   DATA[2383,13] := 817.9794;
   DATA[2383,14] := 1.0;
   DATA[2383,15] := 2.0;
   DATA[2383,16] := 1.0;
   DATA[2383,17] := 1.0;
   DATA[2383,18] := 1.0;
   DATA[2383,19] := 2.0;
   DATA[2383,20] := 148.808;
   DATA[2383,21] := 155.0372;
   DATA[2383,22] := 1.71262;
   DATA[2383,23] := 858.5875;
   DATA[2383,24] := 2.0;
   DATA[2383,25] := 2.0;
   DATA[2383,26] := 7.874135;
   DATA[2383,27] := 144.1938;
   DATA[2383,28] := 261.7278;
   DATA[2383,29] := 12.11228;
   DATA[2383,30] := 1.725711;
   DATA[2383,31] := 1.28705;
   DATA[2383,32] := 0.7353967;
   DATA[2383,33] := 0.3084265;
   DATA[2383,34] := 2.0;
   DATA[2383,35] := 250.0801;
   DATA[2383,36] := 1.681991;
   DATA[2383,37] := 188.7977;
   DATA[2383,38] := 0.000128152;
   DATA[2383,39] := 1.0;
   DATA[2383,40] := 1.0;
   DATA[2384,0] := 2.655414;
   DATA[2384,1] := 865.8766;
   DATA[2384,2] := 2.0;
   DATA[2384,3] := 2.0;
   DATA[2384,4] := 262.3366;
   DATA[2384,5] := 8.395475;
   DATA[2384,6] := 329.7103;
   DATA[2384,7] := 2.455131;
   DATA[2384,8] := 2.0;
   DATA[2384,9] := 2.0;
   DATA[2384,10] := 2.0;
   DATA[2384,11] := 19.66195;
   DATA[2384,12] := 2.208244;
   DATA[2384,13] := 818.0595;
   DATA[2384,14] := 1.0;
   DATA[2384,15] := 2.0;
   DATA[2384,16] := 1.0;
   DATA[2384,17] := 1.0;
   DATA[2384,18] := 1.0;
   DATA[2384,19] := 2.0;
   DATA[2384,20] := 148.808;
   DATA[2384,21] := 155.0372;
   DATA[2384,22] := 1.713901;
   DATA[2384,23] := 858.5491;
   DATA[2384,24] := 2.0;
   DATA[2384,25] := 2.0;
   DATA[2384,26] := 7.874135;
   DATA[2384,27] := 144.1938;
   DATA[2384,28] := 261.7278;
   DATA[2384,29] := 12.11228;
   DATA[2384,30] := 1.725711;
   DATA[2384,31] := 1.277443;
   DATA[2384,32] := 0.7353967;
   DATA[2384,33] := 0.3084265;
   DATA[2384,34] := 2.0;
   DATA[2384,35] := 250.0801;
   DATA[2384,36] := 1.681991;
   DATA[2384,37] := 188.7977;
   DATA[2384,38] := 0.000128152;
   DATA[2384,39] := 1.0;
   DATA[2384,40] := 1.0;
   DATA[2385,0] := 2.653813;
   DATA[2385,1] := 865.9943;
   DATA[2385,2] := 2.0;
   DATA[2385,3] := 2.0;
   DATA[2385,4] := 262.3366;
   DATA[2385,5] := 8.395475;
   DATA[2385,6] := 329.7103;
   DATA[2385,7] := 2.455131;
   DATA[2385,8] := 2.0;
   DATA[2385,9] := 2.0;
   DATA[2385,10] := 2.0;
   DATA[2385,11] := 19.68436;
   DATA[2385,12] := 2.208244;
   DATA[2385,13] := 818.1796;
   DATA[2385,14] := 1.0;
   DATA[2385,15] := 2.0;
   DATA[2385,16] := 1.0;
   DATA[2385,17] := 1.0;
   DATA[2385,18] := 1.0;
   DATA[2385,19] := 2.0;
   DATA[2385,20] := 148.808;
   DATA[2385,21] := 155.0372;
   DATA[2385,22] := 1.713901;
   DATA[2385,23] := 858.7413;
   DATA[2385,24] := 2.0;
   DATA[2385,25] := 2.0;
   DATA[2385,26] := 7.874135;
   DATA[2385,27] := 144.1938;
   DATA[2385,28] := 261.7278;
   DATA[2385,29] := 12.11228;
   DATA[2385,30] := 1.725711;
   DATA[2385,31] := 1.265147;
   DATA[2385,32] := 0.7353967;
   DATA[2385,33] := 0.3084265;
   DATA[2385,34] := 2.0;
   DATA[2385,35] := 249.984;
   DATA[2385,36] := 1.681991;
   DATA[2385,37] := 188.8138;
   DATA[2385,38] := 0.000128152;
   DATA[2385,39] := 1.0;
   DATA[2385,40] := 1.0;
   DATA[2386,0] := 2.625308;
   DATA[2386,1] := 866.5439;
   DATA[2386,2] := 2.0;
   DATA[2386,3] := 2.0;
   DATA[2386,4] := 262.3366;
   DATA[2386,5] := 8.395475;
   DATA[2386,6] := 329.7103;
   DATA[2386,7] := 2.456284;
   DATA[2386,8] := 2.0;
   DATA[2386,9] := 2.0;
   DATA[2386,10] := 2.0;
   DATA[2386,11] := 19.70357;
   DATA[2386,12] := 2.208244;
   DATA[2386,13] := 818.1796;
   DATA[2386,14] := 1.0;
   DATA[2386,15] := 2.0;
   DATA[2386,16] := 1.0;
   DATA[2386,17] := 1.0;
   DATA[2386,18] := 1.0;
   DATA[2386,19] := 2.0;
   DATA[2386,20] := 148.808;
   DATA[2386,21] := 155.0372;
   DATA[2386,22] := 1.713901;
   DATA[2386,23] := 859.0874;
   DATA[2386,24] := 2.0;
   DATA[2386,25] := 2.0;
   DATA[2386,26] := 7.874135;
   DATA[2386,27] := 144.2451;
   DATA[2386,28] := 261.7278;
   DATA[2386,29] := 12.11228;
   DATA[2386,30] := 1.725711;
   DATA[2386,31] := 1.271935;
   DATA[2386,32] := 0.7353967;
   DATA[2386,33] := 0.3084265;
   DATA[2386,34] := 2.0;
   DATA[2386,35] := 249.984;
   DATA[2386,36] := 1.681991;
   DATA[2386,37] := 188.8939;
   DATA[2386,38] := 0.000128152;
   DATA[2386,39] := 1.0;
   DATA[2386,40] := 1.0;
   DATA[2387,0] := 2.612818;
   DATA[2387,1] := 866.7009;
   DATA[2387,2] := 2.0;
   DATA[2387,3] := 2.0;
   DATA[2387,4] := 262.3366;
   DATA[2387,5] := 8.395475;
   DATA[2387,6] := 329.7103;
   DATA[2387,7] := 2.456284;
   DATA[2387,8] := 2.0;
   DATA[2387,9] := 2.0;
   DATA[2387,10] := 2.0;
   DATA[2387,11] := 19.67796;
   DATA[2387,12] := 2.208244;
   DATA[2387,13] := 818.2598;
   DATA[2387,14] := 1.0;
   DATA[2387,15] := 2.0;
   DATA[2387,16] := 1.0;
   DATA[2387,17] := 1.0;
   DATA[2387,18] := 1.0;
   DATA[2387,19] := 2.0;
   DATA[2387,20] := 148.808;
   DATA[2387,21] := 155.0372;
   DATA[2387,22] := 1.714798;
   DATA[2387,23] := 859.2797;
   DATA[2387,24] := 2.0;
   DATA[2387,25] := 2.0;
   DATA[2387,26] := 7.874135;
   DATA[2387,27] := 144.322;
   DATA[2387,28] := 261.7278;
   DATA[2387,29] := 11.95847;
   DATA[2387,30] := 1.725711;
   DATA[2387,31] := 1.279365;
   DATA[2387,32] := 0.7353967;
   DATA[2387,33] := 0.3084265;
   DATA[2387,34] := 2.0;
   DATA[2387,35] := 249.984;
   DATA[2387,36] := 1.681991;
   DATA[2387,37] := 188.8939;
   DATA[2387,38] := 0.000128152;
   DATA[2387,39] := 1.0;
   DATA[2387,40] := 1.0;
   DATA[2388,0] := 2.610575;
   DATA[2388,1] := 867.0542;
   DATA[2388,2] := 2.0;
   DATA[2388,3] := 2.0;
   DATA[2388,4] := 262.3366;
   DATA[2388,5] := 8.395475;
   DATA[2388,6] := 329.7103;
   DATA[2388,7] := 2.456284;
   DATA[2388,8] := 2.0;
   DATA[2388,9] := 2.0;
   DATA[2388,10] := 2.0;
   DATA[2388,11] := 19.62033;
   DATA[2388,12] := 2.206963;
   DATA[2388,13] := 818.1796;
   DATA[2388,14] := 1.0;
   DATA[2388,15] := 2.0;
   DATA[2388,16] := 1.0;
   DATA[2388,17] := 1.0;
   DATA[2388,18] := 1.0;
   DATA[2388,19] := 2.0;
   DATA[2388,20] := 148.808;
   DATA[2388,21] := 155.0372;
   DATA[2388,22] := 1.715952;
   DATA[2388,23] := 859.1643;
   DATA[2388,24] := 2.0;
   DATA[2388,25] := 2.0;
   DATA[2388,26] := 7.874135;
   DATA[2388,27] := 144.4501;
   DATA[2388,28] := 261.7278;
   DATA[2388,29] := 11.95847;
   DATA[2388,30] := 1.725711;
   DATA[2388,31] := 1.282311;
   DATA[2388,32] := 0.7353967;
   DATA[2388,33] := 0.3084265;
   DATA[2388,34] := 2.0;
   DATA[2388,35] := 249.984;
   DATA[2388,36] := 1.681991;
   DATA[2388,37] := 188.8939;
   DATA[2388,38] := 0.000128152;
   DATA[2388,39] := 1.0;
   DATA[2388,40] := 1.0;
   DATA[2389,0] := 2.600967;
   DATA[2389,1] := 867.2504;
   DATA[2389,2] := 2.0;
   DATA[2389,3] := 2.0;
   DATA[2389,4] := 262.3366;
   DATA[2389,5] := 8.395475;
   DATA[2389,6] := 329.7103;
   DATA[2389,7] := 2.455003;
   DATA[2389,8] := 2.0;
   DATA[2389,9] := 2.0;
   DATA[2389,10] := 2.0;
   DATA[2389,11] := 19.62033;
   DATA[2389,12] := 2.206963;
   DATA[2389,13] := 818.2598;
   DATA[2389,14] := 1.0;
   DATA[2389,15] := 2.0;
   DATA[2389,16] := 1.0;
   DATA[2389,17] := 1.0;
   DATA[2389,18] := 1.0;
   DATA[2389,19] := 2.0;
   DATA[2389,20] := 148.808;
   DATA[2389,21] := 155.0372;
   DATA[2389,22] := 1.717105;
   DATA[2389,23] := 859.3566;
   DATA[2389,24] := 2.0;
   DATA[2389,25] := 2.0;
   DATA[2389,26] := 7.874135;
   DATA[2389,27] := 144.4501;
   DATA[2389,28] := 261.5996;
   DATA[2389,29] := 11.95847;
   DATA[2389,30] := 1.725711;
   DATA[2389,31] := 1.288843;
   DATA[2389,32] := 0.7353967;
   DATA[2389,33] := 0.3084265;
   DATA[2389,34] := 2.0;
   DATA[2389,35] := 249.984;
   DATA[2389,36] := 1.681991;
   DATA[2389,37] := 188.8939;
   DATA[2389,38] := 0.000128152;
   DATA[2389,39] := 1.0;
   DATA[2389,40] := 1.0;
   DATA[2390,0] := 2.600967;
   DATA[2390,1] := 867.2504;
   DATA[2390,2] := 2.0;
   DATA[2390,3] := 2.0;
   DATA[2390,4] := 262.3366;
   DATA[2390,5] := 8.395475;
   DATA[2390,6] := 329.7103;
   DATA[2390,7] := 2.455003;
   DATA[2390,8] := 2.0;
   DATA[2390,9] := 2.0;
   DATA[2390,10] := 2.0;
   DATA[2390,11] := 19.62033;
   DATA[2390,12] := 2.206963;
   DATA[2390,13] := 818.2598;
   DATA[2390,14] := 1.0;
   DATA[2390,15] := 2.0;
   DATA[2390,16] := 1.0;
   DATA[2390,17] := 1.0;
   DATA[2390,18] := 1.0;
   DATA[2390,19] := 2.0;
   DATA[2390,20] := 148.808;
   DATA[2390,21] := 155.0372;
   DATA[2390,22] := 1.717105;
   DATA[2390,23] := 859.3566;
   DATA[2390,24] := 2.0;
   DATA[2390,25] := 2.0;
   DATA[2390,26] := 7.874135;
   DATA[2390,27] := 144.4501;
   DATA[2390,28] := 261.5996;
   DATA[2390,29] := 11.95847;
   DATA[2390,30] := 1.725711;
   DATA[2390,31] := 1.288843;
   DATA[2390,32] := 0.7353967;
   DATA[2390,33] := 0.3084265;
   DATA[2390,34] := 2.0;
   DATA[2390,35] := 249.984;
   DATA[2390,36] := 1.681991;
   DATA[2390,37] := 188.8939;
   DATA[2390,38] := 0.000128152;
   DATA[2390,39] := 1.0;
   DATA[2390,40] := 1.0;
   DATA[2391,0] := 2.578548;
   DATA[2391,1] := 867.2504;
   DATA[2391,2] := 2.0;
   DATA[2391,3] := 2.0;
   DATA[2391,4] := 262.3366;
   DATA[2391,5] := 8.395475;
   DATA[2391,6] := 329.7103;
   DATA[2391,7] := 2.454362;
   DATA[2391,8] := 2.0;
   DATA[2391,9] := 2.0;
   DATA[2391,10] := 2.0;
   DATA[2391,11] := 19.62994;
   DATA[2391,12] := 2.206963;
   DATA[2391,13] := 818.3398;
   DATA[2391,14] := 1.0;
   DATA[2391,15] := 2.0;
   DATA[2391,16] := 1.0;
   DATA[2391,17] := 1.0;
   DATA[2391,18] := 1.0;
   DATA[2391,19] := 2.0;
   DATA[2391,20] := 148.808;
   DATA[2391,21] := 155.0372;
   DATA[2391,22] := 1.717361;
   DATA[2391,23] := 859.5873;
   DATA[2391,24] := 2.0;
   DATA[2391,25] := 2.0;
   DATA[2391,26] := 7.874135;
   DATA[2391,27] := 144.4501;
   DATA[2391,28] := 261.5996;
   DATA[2391,29] := 11.95847;
   DATA[2391,30] := 1.725711;
   DATA[2391,31] := 1.291789;
   DATA[2391,32] := 0.7353967;
   DATA[2391,33] := 0.3084265;
   DATA[2391,34] := 2.0;
   DATA[2391,35] := 250.1602;
   DATA[2391,36] := 1.681991;
   DATA[2391,37] := 188.8939;
   DATA[2391,38] := 0.000128152;
   DATA[2391,39] := 1.0;
   DATA[2391,40] := 1.0;
   DATA[2392,0] := 2.564135;
   DATA[2392,1] := 867.3289;
   DATA[2392,2] := 2.0;
   DATA[2392,3] := 2.0;
   DATA[2392,4] := 262.3366;
   DATA[2392,5] := 8.395475;
   DATA[2392,6] := 329.7103;
   DATA[2392,7] := 2.454362;
   DATA[2392,8] := 2.0;
   DATA[2392,9] := 2.0;
   DATA[2392,10] := 2.0;
   DATA[2392,11] := 19.66835;
   DATA[2392,12] := 2.206963;
   DATA[2392,13] := 818.1396;
   DATA[2392,14] := 1.0;
   DATA[2392,15] := 2.0;
   DATA[2392,16] := 1.0;
   DATA[2392,17] := 1.0;
   DATA[2392,18] := 1.0;
   DATA[2392,19] := 2.0;
   DATA[2392,20] := 148.808;
   DATA[2392,21] := 155.191;
   DATA[2392,22] := 1.718643;
   DATA[2392,23] := 859.5873;
   DATA[2392,24] := 2.0;
   DATA[2392,25] := 2.0;
   DATA[2392,26] := 7.874135;
   DATA[2392,27] := 144.4501;
   DATA[2392,28] := 261.5996;
   DATA[2392,29] := 11.95847;
   DATA[2392,30] := 1.725711;
   DATA[2392,31] := 1.291405;
   DATA[2392,32] := 0.7353967;
   DATA[2392,33] := 0.3084265;
   DATA[2392,34] := 2.0;
   DATA[2392,35] := 250.1602;
   DATA[2392,36] := 1.681991;
   DATA[2392,37] := 188.8939;
   DATA[2392,38] := 0.000128152;
   DATA[2392,39] := 1.0;
   DATA[2392,40] := 1.0;
   DATA[2393,0] := 2.54684;
   DATA[2393,1] := 867.3289;
   DATA[2393,2] := 2.0;
   DATA[2393,3] := 2.0;
   DATA[2393,4] := 262.3366;
   DATA[2393,5] := 8.395475;
   DATA[2393,6] := 329.7103;
   DATA[2393,7] := 2.454362;
   DATA[2393,8] := 2.0;
   DATA[2393,9] := 2.0;
   DATA[2393,10] := 2.0;
   DATA[2393,11] := 19.66835;
   DATA[2393,12] := 2.206963;
   DATA[2393,13] := 818.2197;
   DATA[2393,14] := 1.0;
   DATA[2393,15] := 2.0;
   DATA[2393,16] := 1.0;
   DATA[2393,17] := 1.0;
   DATA[2393,18] := 1.0;
   DATA[2393,19] := 2.0;
   DATA[2393,20] := 148.808;
   DATA[2393,21] := 155.191;
   DATA[2393,22] := 1.718643;
   DATA[2393,23] := 859.395;
   DATA[2393,24] := 2.0;
   DATA[2393,25] := 2.0;
   DATA[2393,26] := 7.874135;
   DATA[2393,27] := 144.4501;
   DATA[2393,28] := 261.5996;
   DATA[2393,29] := 11.95847;
   DATA[2393,30] := 1.725711;
   DATA[2393,31] := 1.283592;
   DATA[2393,32] := 0.7353967;
   DATA[2393,33] := 0.3084265;
   DATA[2393,34] := 2.0;
   DATA[2393,35] := 250.1602;
   DATA[2393,36] := 1.681991;
   DATA[2393,37] := 188.8939;
   DATA[2393,38] := 0.000128152;
   DATA[2393,39] := 1.0;
   DATA[2393,40] := 1.0;
   DATA[2394,0] := 2.533068;
   DATA[2394,1] := 867.3289;
   DATA[2394,2] := 2.0;
   DATA[2394,3] := 2.0;
   DATA[2394,4] := 262.3366;
   DATA[2394,5] := 8.395475;
   DATA[2394,6] := 329.7103;
   DATA[2394,7] := 2.45449;
   DATA[2394,8] := 2.0;
   DATA[2394,9] := 2.0;
   DATA[2394,10] := 2.0;
   DATA[2394,11] := 19.66835;
   DATA[2394,12] := 2.208372;
   DATA[2394,13] := 818.3398;
   DATA[2394,14] := 1.0;
   DATA[2394,15] := 2.0;
   DATA[2394,16] := 1.0;
   DATA[2394,17] := 1.0;
   DATA[2394,18] := 1.0;
   DATA[2394,19] := 2.0;
   DATA[2394,20] := 148.808;
   DATA[2394,21] := 155.191;
   DATA[2394,22] := 1.718643;
   DATA[2394,23] := 859.8564;
   DATA[2394,24] := 2.0;
   DATA[2394,25] := 2.0;
   DATA[2394,26] := 7.874135;
   DATA[2394,27] := 144.4501;
   DATA[2394,28] := 261.5996;
   DATA[2394,29] := 11.95847;
   DATA[2394,30] := 1.725711;
   DATA[2394,31] := 1.273601;
   DATA[2394,32] := 0.7353967;
   DATA[2394,33] := 0.3084265;
   DATA[2394,34] := 2.0;
   DATA[2394,35] := 250.1602;
   DATA[2394,36] := 1.617916;
   DATA[2394,37] := 188.8939;
   DATA[2394,38] := 0.000128152;
   DATA[2394,39] := 1.0;
   DATA[2394,40] := 1.0;
   DATA[2395,0] := 2.516414;
   DATA[2395,1] := 867.3289;
   DATA[2395,2] := 2.0;
   DATA[2395,3] := 2.0;
   DATA[2395,4] := 262.3366;
   DATA[2395,5] := 8.395475;
   DATA[2395,6] := 329.7103;
   DATA[2395,7] := 2.45449;
   DATA[2395,8] := 2.0;
   DATA[2395,9] := 2.0;
   DATA[2395,10] := 2.0;
   DATA[2395,11] := 19.67796;
   DATA[2395,12] := 2.209397;
   DATA[2395,13] := 818.8205;
   DATA[2395,14] := 1.0;
   DATA[2395,15] := 2.0;
   DATA[2395,16] := 1.0;
   DATA[2395,17] := 1.0;
   DATA[2395,18] := 1.0;
   DATA[2395,19] := 2.0;
   DATA[2395,20] := 148.808;
   DATA[2395,21] := 155.191;
   DATA[2395,22] := 1.718643;
   DATA[2395,23] := 859.9718;
   DATA[2395,24] := 2.0;
   DATA[2395,25] := 2.0;
   DATA[2395,26] := 7.874135;
   DATA[2395,27] := 144.4501;
   DATA[2395,28] := 261.5996;
   DATA[2395,29] := 11.95847;
   DATA[2395,30] := 1.725711;
   DATA[2395,31] := 1.264378;
   DATA[2395,32] := 0.7353967;
   DATA[2395,33] := 0.3084265;
   DATA[2395,34] := 2.0;
   DATA[2395,35] := 250.1602;
   DATA[2395,36] := 1.617916;
   DATA[2395,37] := 188.8939;
   DATA[2395,38] := 0.000128152;
   DATA[2395,39] := 1.0;
   DATA[2395,40] := 1.0;
   DATA[2396,0] := 2.503283;
   DATA[2396,1] := 867.3682;
   DATA[2396,2] := 2.0;
   DATA[2396,3] := 2.0;
   DATA[2396,4] := 262.3366;
   DATA[2396,5] := 8.395475;
   DATA[2396,6] := 329.7103;
   DATA[2396,7] := 2.45449;
   DATA[2396,8] := 2.0;
   DATA[2396,9] := 2.0;
   DATA[2396,10] := 2.0;
   DATA[2396,11] := 19.70997;
   DATA[2396,12] := 2.209397;
   DATA[2396,13] := 819.1409;
   DATA[2396,14] := 1.0;
   DATA[2396,15] := 2.0;
   DATA[2396,16] := 1.0;
   DATA[2396,17] := 1.0;
   DATA[2396,18] := 1.0;
   DATA[2396,19] := 2.0;
   DATA[2396,20] := 148.808;
   DATA[2396,21] := 155.191;
   DATA[2396,22] := 1.718643;
   DATA[2396,23] := 859.8564;
   DATA[2396,24] := 2.0;
   DATA[2396,25] := 2.0;
   DATA[2396,26] := 7.874135;
   DATA[2396,27] := 144.4501;
   DATA[2396,28] := 261.5996;
   DATA[2396,29] := 11.95847;
   DATA[2396,30] := 1.725711;
   DATA[2396,31] := 1.261688;
   DATA[2396,32] := 0.7353967;
   DATA[2396,33] := 0.3084265;
   DATA[2396,34] := 2.0;
   DATA[2396,35] := 250.1602;
   DATA[2396,36] := 1.617916;
   DATA[2396,37] := 188.8939;
   DATA[2396,38] := 0.000128152;
   DATA[2396,39] := 1.0;
   DATA[2396,40] := 1.0;
   DATA[2397,0] := 2.481504;
   DATA[2397,1] := 867.2897;
   DATA[2397,2] := 2.0;
   DATA[2397,3] := 2.0;
   DATA[2397,4] := 262.3366;
   DATA[2397,5] := 8.395475;
   DATA[2397,6] := 329.7103;
   DATA[2397,7] := 2.45449;
   DATA[2397,8] := 2.0;
   DATA[2397,9] := 2.0;
   DATA[2397,10] := 2.0;
   DATA[2397,11] := 19.70997;
   DATA[2397,12] := 2.210678;
   DATA[2397,13] := 819.0609;
   DATA[2397,14] := 1.0;
   DATA[2397,15] := 2.0;
   DATA[2397,16] := 1.0;
   DATA[2397,17] := 1.0;
   DATA[2397,18] := 1.0;
   DATA[2397,19] := 2.0;
   DATA[2397,20] := 148.808;
   DATA[2397,21] := 155.191;
   DATA[2397,22] := 1.718643;
   DATA[2397,23] := 859.7795;
   DATA[2397,24] := 2.0;
   DATA[2397,25] := 2.0;
   DATA[2397,26] := 7.874135;
   DATA[2397,27] := 144.4501;
   DATA[2397,28] := 261.5996;
   DATA[2397,29] := 11.95847;
   DATA[2397,30] := 1.725711;
   DATA[2397,31] := 1.267709;
   DATA[2397,32] := 0.7353967;
   DATA[2397,33] := 0.3084265;
   DATA[2397,34] := 2.0;
   DATA[2397,35] := 250.1602;
   DATA[2397,36] := 1.617916;
   DATA[2397,37] := 188.8939;
   DATA[2397,38] := 0.000128152;
   DATA[2397,39] := 1.0;
   DATA[2397,40] := 1.0;
   DATA[2398,0] := 2.469013;
   DATA[2398,1] := 867.5645;
   DATA[2398,2] := 2.0;
   DATA[2398,3] := 2.0;
   DATA[2398,4] := 262.3366;
   DATA[2398,5] := 8.395475;
   DATA[2398,6] := 329.7103;
   DATA[2398,7] := 2.45449;
   DATA[2398,8] := 2.0;
   DATA[2398,9] := 2.0;
   DATA[2398,10] := 2.0;
   DATA[2398,11] := 19.70997;
   DATA[2398,12] := 2.210806;
   DATA[2398,13] := 819.181;
   DATA[2398,14] := 1.0;
   DATA[2398,15] := 2.0;
   DATA[2398,16] := 1.0;
   DATA[2398,17] := 1.0;
   DATA[2398,18] := 1.0;
   DATA[2398,19] := 2.0;
   DATA[2398,20] := 148.808;
   DATA[2398,21] := 155.191;
   DATA[2398,22] := 1.718643;
   DATA[2398,23] := 859.1643;
   DATA[2398,24] := 2.0;
   DATA[2398,25] := 2.0;
   DATA[2398,26] := 7.874135;
   DATA[2398,27] := 144.4501;
   DATA[2398,28] := 261.5996;
   DATA[2398,29] := 11.95847;
   DATA[2398,30] := 1.725711;
   DATA[2398,31] := 1.261688;
   DATA[2398,32] := 0.7353967;
   DATA[2398,33] := 0.3084265;
   DATA[2398,34] := 2.0;
   DATA[2398,35] := 250.1602;
   DATA[2398,36] := 1.617916;
   DATA[2398,37] := 188.8939;
   DATA[2398,38] := 0.000128152;
   DATA[2398,39] := 1.0;
   DATA[2398,40] := 1.0;
   DATA[2399,0] := 2.44243;
   DATA[2399,1] := 866.9756;
   DATA[2399,2] := 2.0;
   DATA[2399,3] := 2.0;
   DATA[2399,4] := 262.3366;
   DATA[2399,5] := 8.395475;
   DATA[2399,6] := 329.7103;
   DATA[2399,7] := 2.45449;
   DATA[2399,8] := 2.0;
   DATA[2399,9] := 2.0;
   DATA[2399,10] := 2.0;
   DATA[2399,11] := 19.70997;
   DATA[2399,12] := 2.210806;
   DATA[2399,13] := 819.5415;
   DATA[2399,14] := 1.0;
   DATA[2399,15] := 2.0;
   DATA[2399,16] := 1.0;
   DATA[2399,17] := 1.0;
   DATA[2399,18] := 1.0;
   DATA[2399,19] := 2.0;
   DATA[2399,20] := 148.808;
   DATA[2399,21] := 155.191;
   DATA[2399,22] := 1.718643;
   DATA[2399,23] := 858.8951;
   DATA[2399,24] := 2.0;
   DATA[2399,25] := 2.0;
   DATA[2399,26] := 7.874135;
   DATA[2399,27] := 144.4501;
   DATA[2399,28] := 261.5996;
   DATA[2399,29] := 11.95847;
   DATA[2399,30] := 1.725968;
   DATA[2399,31] := 1.263866;
   DATA[2399,32] := 0.7353967;
   DATA[2399,33] := 0.3084265;
   DATA[2399,34] := 2.0;
   DATA[2399,35] := 250.0;
   DATA[2399,36] := 1.69801;
   DATA[2399,37] := 188.8939;
   DATA[2399,38] := 0.000128152;
   DATA[2399,39] := 1.0;
   DATA[2399,40] := 1.0;
   DATA[2400,0] := 2.431221;
   DATA[2400,1] := 867.0934;
   DATA[2400,2] := 2.0;
   DATA[2400,3] := 2.0;
   DATA[2400,4] := 262.3366;
   DATA[2400,5] := 8.395475;
   DATA[2400,6] := 329.8129;
   DATA[2400,7] := 2.45449;
   DATA[2400,8] := 2.0;
   DATA[2400,9] := 2.0;
   DATA[2400,10] := 2.0;
   DATA[2400,11] := 19.70997;
   DATA[2400,12] := 2.210806;
   DATA[2400,13] := 819.5815;
   DATA[2400,14] := 1.0;
   DATA[2400,15] := 2.0;
   DATA[2400,16] := 1.0;
   DATA[2400,17] := 1.0;
   DATA[2400,18] := 1.0;
   DATA[2400,19] := 2.0;
   DATA[2400,20] := 148.808;
   DATA[2400,21] := 155.191;
   DATA[2400,22] := 1.718643;
   DATA[2400,23] := 858.972;
   DATA[2400,24] := 2.0;
   DATA[2400,25] := 2.0;
   DATA[2400,26] := 7.874135;
   DATA[2400,27] := 144.4501;
   DATA[2400,28] := 261.5996;
   DATA[2400,29] := 11.95847;
   DATA[2400,30] := 1.726352;
   DATA[2400,31] := 1.271295;
   DATA[2400,32] := 0.7353967;
   DATA[2400,33] := 0.3084265;
   DATA[2400,34] := 2.0;
   DATA[2400,35] := 249.9359;
   DATA[2400,36] := 1.69801;
   DATA[2400,37] := 188.8939;
   DATA[2400,38] := 0.000128152;
   DATA[2400,39] := 1.0;
   DATA[2400,40] := 1.0;
   DATA[2401,0] := 2.428018;
   DATA[2401,1] := 866.6616;
   DATA[2401,2] := 2.0;
   DATA[2401,3] := 2.0;
   DATA[2401,4] := 262.3366;
   DATA[2401,5] := 8.395475;
   DATA[2401,6] := 329.8129;
   DATA[2401,7] := 2.45449;
   DATA[2401,8] := 2.0;
   DATA[2401,9] := 2.0;
   DATA[2401,10] := 2.0;
   DATA[2401,11] := 19.70997;
   DATA[2401,12] := 2.210806;
   DATA[2401,13] := 819.3412;
   DATA[2401,14] := 1.0;
   DATA[2401,15] := 2.0;
   DATA[2401,16] := 1.0;
   DATA[2401,17] := 1.0;
   DATA[2401,18] := 1.0;
   DATA[2401,19] := 2.0;
   DATA[2401,20] := 148.808;
   DATA[2401,21] := 155.191;
   DATA[2401,22] := 1.717233;
   DATA[2401,23] := 858.972;
   DATA[2401,24] := 2.0;
   DATA[2401,25] := 2.0;
   DATA[2401,26] := 7.874135;
   DATA[2401,27] := 144.4501;
   DATA[2401,28] := 261.5996;
   DATA[2401,29] := 11.95847;
   DATA[2401,30] := 1.726352;
   DATA[2401,31] := 1.285001;
   DATA[2401,32] := 0.7353967;
   DATA[2401,33] := 0.3084265;
   DATA[2401,34] := 2.0;
   DATA[2401,35] := 249.9359;
   DATA[2401,36] := 1.69801;
   DATA[2401,37] := 188.8939;
   DATA[2401,38] := 0.000128152;
   DATA[2401,39] := 1.0;
   DATA[2401,40] := 1.0;
   DATA[2402,0] := 2.428018;
   DATA[2402,1] := 866.8579;
   DATA[2402,2] := 2.0;
   DATA[2402,3] := 2.0;
   DATA[2402,4] := 262.3366;
   DATA[2402,5] := 8.395475;
   DATA[2402,6] := 329.8129;
   DATA[2402,7] := 2.45449;
   DATA[2402,8] := 2.0;
   DATA[2402,9] := 2.0;
   DATA[2402,10] := 2.0;
   DATA[2402,11] := 19.70997;
   DATA[2402,12] := 2.210806;
   DATA[2402,13] := 819.7818;
   DATA[2402,14] := 1.0;
   DATA[2402,15] := 2.0;
   DATA[2402,16] := 1.0;
   DATA[2402,17] := 1.0;
   DATA[2402,18] := 1.0;
   DATA[2402,19] := 2.0;
   DATA[2402,20] := 148.808;
   DATA[2402,21] := 155.191;
   DATA[2402,22] := 1.714926;
   DATA[2402,23] := 858.8182;
   DATA[2402,24] := 2.0;
   DATA[2402,25] := 2.0;
   DATA[2402,26] := 7.874135;
   DATA[2402,27] := 144.4501;
   DATA[2402,28] := 261.5996;
   DATA[2402,29] := 11.95847;
   DATA[2402,30] := 1.726224;
   DATA[2402,31] := 1.301012;
   DATA[2402,32] := 0.7353967;
   DATA[2402,33] := 0.3084265;
   DATA[2402,34] := 2.0;
   DATA[2402,35] := 249.9359;
   DATA[2402,36] := 1.69801;
   DATA[2402,37] := 188.6375;
   DATA[2402,38] := 0.000128152;
   DATA[2402,39] := 1.0;
   DATA[2402,40] := 1.0;
   DATA[2403,0] := 2.448836;
   DATA[2403,1] := 866.5439;
   DATA[2403,2] := 2.0;
   DATA[2403,3] := 2.0;
   DATA[2403,4] := 262.3366;
   DATA[2403,5] := 8.395475;
   DATA[2403,6] := 329.8129;
   DATA[2403,7] := 2.455515;
   DATA[2403,8] := 2.0;
   DATA[2403,9] := 2.0;
   DATA[2403,10] := 2.0;
   DATA[2403,11] := 19.71957;
   DATA[2403,12] := 2.210806;
   DATA[2403,13] := 819.8218;
   DATA[2403,14] := 1.0;
   DATA[2403,15] := 2.0;
   DATA[2403,16] := 1.0;
   DATA[2403,17] := 1.0;
   DATA[2403,18] := 1.0;
   DATA[2403,19] := 2.0;
   DATA[2403,20] := 148.808;
   DATA[2403,21] := 155.191;
   DATA[2403,22] := 1.713517;
   DATA[2403,23] := 859.0874;
   DATA[2403,24] := 2.0;
   DATA[2403,25] := 2.0;
   DATA[2403,26] := 7.874135;
   DATA[2403,27] := 144.4501;
   DATA[2403,28] := 261.5996;
   DATA[2403,29] := 11.95847;
   DATA[2403,30] := 1.724942;
   DATA[2403,31] := 1.30178;
   DATA[2403,32] := 0.7353967;
   DATA[2403,33] := 0.3084265;
   DATA[2403,34] := 2.0;
   DATA[2403,35] := 249.8718;
   DATA[2403,36] := 1.69801;
   DATA[2403,37] := 188.6375;
   DATA[2403,38] := 0.000128152;
   DATA[2403,39] := 1.0;
   DATA[2403,40] := 1.0;
   DATA[2404,0] := 2.494315;
   DATA[2404,1] := 866.5439;
   DATA[2404,2] := 2.0;
   DATA[2404,3] := 2.0;
   DATA[2404,4] := 262.3366;
   DATA[2404,5] := 8.395475;
   DATA[2404,6] := 329.8129;
   DATA[2404,7] := 2.456284;
   DATA[2404,8] := 2.0;
   DATA[2404,9] := 2.0;
   DATA[2404,10] := 2.0;
   DATA[2404,11] := 19.76439;
   DATA[2404,12] := 2.210037;
   DATA[2404,13] := 820.1824;
   DATA[2404,14] := 1.0;
   DATA[2404,15] := 2.0;
   DATA[2404,16] := 1.0;
   DATA[2404,17] := 1.0;
   DATA[2404,18] := 1.0;
   DATA[2404,19] := 2.0;
   DATA[2404,20] := 148.808;
   DATA[2404,21] := 155.191;
   DATA[2404,22] := 1.713517;
   DATA[2404,23] := 858.7413;
   DATA[2404,24] := 2.0;
   DATA[2404,25] := 2.0;
   DATA[2404,26] := 7.874135;
   DATA[2404,27] := 144.4501;
   DATA[2404,28] := 261.5996;
   DATA[2404,29] := 11.95847;
   DATA[2404,30] := 1.722892;
   DATA[2404,31] := 1.296401;
   DATA[2404,32] := 0.7353967;
   DATA[2404,33] := 0.3084265;
   DATA[2404,34] := 2.0;
   DATA[2404,35] := 249.7116;
   DATA[2404,36] := 1.69801;
   DATA[2404,37] := 188.6375;
   DATA[2404,38] := 0.000128152;
   DATA[2404,39] := 1.0;
   DATA[2404,40] := 1.0;
   DATA[2405,0] := 2.540115;
   DATA[2405,1] := 866.1121;
   DATA[2405,2] := 2.0;
   DATA[2405,3] := 2.0;
   DATA[2405,4] := 262.3366;
   DATA[2405,5] := 8.395475;
   DATA[2405,6] := 329.8129;
   DATA[2405,7] := 2.456284;
   DATA[2405,8] := 2.0;
   DATA[2405,9] := 2.0;
   DATA[2405,10] := 2.0;
   DATA[2405,11] := 19.76439;
   DATA[2405,12] := 2.208756;
   DATA[2405,13] := 820.2224;
   DATA[2405,14] := 1.0;
   DATA[2405,15] := 2.0;
   DATA[2405,16] := 1.0;
   DATA[2405,17] := 1.0;
   DATA[2405,18] := 1.0;
   DATA[2405,19] := 2.0;
   DATA[2405,20] := 148.808;
   DATA[2405,21] := 155.191;
   DATA[2405,22] := 1.713517;
   DATA[2405,23] := 858.7413;
   DATA[2405,24] := 2.0;
   DATA[2405,25] := 2.0;
   DATA[2405,26] := 7.874135;
   DATA[2405,27] := 144.4501;
   DATA[2405,28] := 261.5996;
   DATA[2405,29] := 11.95847;
   DATA[2405,30] := 1.722892;
   DATA[2405,31] := 1.297682;
   DATA[2405,32] := 0.7353967;
   DATA[2405,33] := 0.3084265;
   DATA[2405,34] := 2.0;
   DATA[2405,35] := 249.7116;
   DATA[2405,36] := 1.69801;
   DATA[2405,37] := 188.6375;
   DATA[2405,38] := 0.000128152;
   DATA[2405,39] := 1.0;
   DATA[2405,40] := 1.0;
   DATA[2406,0] := 2.575986;
   DATA[2406,1] := 865.7981;
   DATA[2406,2] := 2.0;
   DATA[2406,3] := 2.0;
   DATA[2406,4] := 262.3366;
   DATA[2406,5] := 8.395475;
   DATA[2406,6] := 329.6591;
   DATA[2406,7] := 2.456284;
   DATA[2406,8] := 2.0;
   DATA[2406,9] := 2.0;
   DATA[2406,10] := 2.0;
   DATA[2406,11] := 19.76439;
   DATA[2406,12] := 2.208628;
   DATA[2406,13] := 820.3826;
   DATA[2406,14] := 1.0;
   DATA[2406,15] := 2.0;
   DATA[2406,16] := 1.0;
   DATA[2406,17] := 1.0;
   DATA[2406,18] := 1.0;
   DATA[2406,19] := 2.0;
   DATA[2406,20] := 148.808;
   DATA[2406,21] := 155.191;
   DATA[2406,22] := 1.712748;
   DATA[2406,23] := 858.7413;
   DATA[2406,24] := 2.0;
   DATA[2406,25] := 2.0;
   DATA[2406,26] := 7.874135;
   DATA[2406,27] := 144.4501;
   DATA[2406,28] := 261.5996;
   DATA[2406,29] := 11.95847;
   DATA[2406,30] := 1.722892;
   DATA[2406,31] := 1.290509;
   DATA[2406,32] := 0.7353967;
   DATA[2406,33] := 0.3084265;
   DATA[2406,34] := 2.0;
   DATA[2406,35] := 249.7116;
   DATA[2406,36] := 1.69801;
   DATA[2406,37] := 188.6375;
   DATA[2406,38] := 0.000128152;
   DATA[2406,39] := 1.0;
   DATA[2406,40] := 1.0;
   DATA[2407,0] := 2.618582;
   DATA[2407,1] := 865.9943;
   DATA[2407,2] := 2.0;
   DATA[2407,3] := 2.0;
   DATA[2407,4] := 262.3366;
   DATA[2407,5] := 8.394514;
   DATA[2407,6] := 329.6591;
   DATA[2407,7] := 2.456284;
   DATA[2407,8] := 2.0;
   DATA[2407,9] := 2.0;
   DATA[2407,10] := 2.0;
   DATA[2407,11] := 19.7996;
   DATA[2407,12] := 2.205041;
   DATA[2407,13] := 820.4627;
   DATA[2407,14] := 1.0;
   DATA[2407,15] := 2.0;
   DATA[2407,16] := 1.0;
   DATA[2407,17] := 1.0;
   DATA[2407,18] := 1.0;
   DATA[2407,19] := 2.0;
   DATA[2407,20] := 148.808;
   DATA[2407,21] := 155.191;
   DATA[2407,22] := 1.712748;
   DATA[2407,23] := 858.5875;
   DATA[2407,24] := 2.0;
   DATA[2407,25] := 2.0;
   DATA[2407,26] := 7.874135;
   DATA[2407,27] := 144.4501;
   DATA[2407,28] := 261.5996;
   DATA[2407,29] := 11.95847;
   DATA[2407,30] := 1.723148;
   DATA[2407,31] := 1.298962;
   DATA[2407,32] := 0.7353967;
   DATA[2407,33] := 0.3084265;
   DATA[2407,34] := 2.0;
   DATA[2407,35] := 249.7116;
   DATA[2407,36] := 1.69801;
   DATA[2407,37] := 188.6375;
   DATA[2407,38] := 0.000128152;
   DATA[2407,39] := 1.0;
   DATA[2407,40] := 1.0;
   DATA[2408,0] := 2.655735;
   DATA[2408,1] := 865.9943;
   DATA[2408,2] := 2.0;
   DATA[2408,3] := 2.0;
   DATA[2408,4] := 262.3366;
   DATA[2408,5] := 8.394514;
   DATA[2408,6] := 329.6591;
   DATA[2408,7] := 2.456284;
   DATA[2408,8] := 2.0;
   DATA[2408,9] := 2.0;
   DATA[2408,10] := 2.0;
   DATA[2408,11] := 19.80601;
   DATA[2408,12] := 2.205041;
   DATA[2408,13] := 820.2625;
   DATA[2408,14] := 1.0;
   DATA[2408,15] := 2.0;
   DATA[2408,16] := 1.0;
   DATA[2408,17] := 1.0;
   DATA[2408,18] := 1.0;
   DATA[2408,19] := 2.0;
   DATA[2408,20] := 148.808;
   DATA[2408,21] := 155.3448;
   DATA[2408,22] := 1.712748;
   DATA[2408,23] := 858.4337;
   DATA[2408,24] := 2.0;
   DATA[2408,25] := 2.0;
   DATA[2408,26] := 7.874135;
   DATA[2408,27] := 144.4501;
   DATA[2408,28] := 261.5996;
   DATA[2408,29] := 11.95847;
   DATA[2408,30] := 1.724301;
   DATA[2408,31] := 1.292686;
   DATA[2408,32] := 0.7353967;
   DATA[2408,33] := 0.3084265;
   DATA[2408,34] := 2.0;
   DATA[2408,35] := 249.8718;
   DATA[2408,36] := 1.69801;
   DATA[2408,37] := 188.6375;
   DATA[2408,38] := 0.000128152;
   DATA[2408,39] := 1.0;
   DATA[2408,40] := 1.0;
   DATA[2409,0] := 2.658937;
   DATA[2409,1] := 866.4654;
   DATA[2409,2] := 2.0;
   DATA[2409,3] := 2.0;
   DATA[2409,4] := 262.3366;
   DATA[2409,5] := 8.394514;
   DATA[2409,6] := 329.6591;
   DATA[2409,7] := 2.456284;
   DATA[2409,8] := 2.0;
   DATA[2409,9] := 2.0;
   DATA[2409,10] := 2.0;
   DATA[2409,11] := 19.80601;
   DATA[2409,12] := 2.205041;
   DATA[2409,13] := 820.0622;
   DATA[2409,14] := 1.0;
   DATA[2409,15] := 2.0;
   DATA[2409,16] := 1.0;
   DATA[2409,17] := 1.0;
   DATA[2409,18] := 1.0;
   DATA[2409,19] := 2.0;
   DATA[2409,20] := 148.808;
   DATA[2409,21] := 155.3448;
   DATA[2409,22] := 1.714798;
   DATA[2409,23] := 858.2415;
   DATA[2409,24] := 2.0;
   DATA[2409,25] := 2.0;
   DATA[2409,26] := 7.874135;
   DATA[2409,27] := 144.4501;
   DATA[2409,28] := 261.5996;
   DATA[2409,29] := 11.95847;
   DATA[2409,30] := 1.724301;
   DATA[2409,31] := 1.282567;
   DATA[2409,32] := 0.7353967;
   DATA[2409,33] := 0.3084265;
   DATA[2409,34] := 2.0;
   DATA[2409,35] := 249.8718;
   DATA[2409,36] := 1.69801;
   DATA[2409,37] := 188.6856;
   DATA[2409,38] := 0.000128152;
   DATA[2409,39] := 1.0;
   DATA[2409,40] := 1.0;
   DATA[2410,0] := 2.646767;
   DATA[2410,1] := 866.5439;
   DATA[2410,2] := 2.0;
   DATA[2410,3] := 2.0;
   DATA[2410,4] := 262.3366;
   DATA[2410,5] := 8.394514;
   DATA[2410,6] := 329.6591;
   DATA[2410,7] := 2.456284;
   DATA[2410,8] := 2.0;
   DATA[2410,9] := 2.0;
   DATA[2410,10] := 2.0;
   DATA[2410,11] := 19.80601;
   DATA[2410,12] := 2.205041;
   DATA[2410,13] := 820.1423;
   DATA[2410,14] := 1.0;
   DATA[2410,15] := 2.0;
   DATA[2410,16] := 1.0;
   DATA[2410,17] := 1.0;
   DATA[2410,18] := 1.0;
   DATA[2410,19] := 2.0;
   DATA[2410,20] := 148.808;
   DATA[2410,21] := 155.3448;
   DATA[2410,22] := 1.715311;
   DATA[2410,23] := 859.1643;
   DATA[2410,24] := 2.0;
   DATA[2410,25] := 2.0;
   DATA[2410,26] := 7.874135;
   DATA[2410,27] := 144.4501;
   DATA[2410,28] := 261.5996;
   DATA[2410,29] := 11.95847;
   DATA[2410,30] := 1.724301;
   DATA[2410,31] := 1.281286;
   DATA[2410,32] := 0.7353967;
   DATA[2410,33] := 0.3084265;
   DATA[2410,34] := 2.0;
   DATA[2410,35] := 249.8718;
   DATA[2410,36] := 1.69801;
   DATA[2410,37] := 188.7657;
   DATA[2410,38] := 0.000128152;
   DATA[2410,39] := 1.0;
   DATA[2410,40] := 1.0;
   DATA[2411,0] := 2.62723;
   DATA[2411,1] := 866.1906;
   DATA[2411,2] := 2.0;
   DATA[2411,3] := 2.0;
   DATA[2411,4] := 262.3366;
   DATA[2411,5] := 8.394514;
   DATA[2411,6] := 329.6591;
   DATA[2411,7] := 2.456284;
   DATA[2411,8] := 2.0;
   DATA[2411,9] := 2.0;
   DATA[2411,10] := 2.0;
   DATA[2411,11] := 19.7804;
   DATA[2411,12] := 2.205554;
   DATA[2411,13] := 820.1423;
   DATA[2411,14] := 1.0;
   DATA[2411,15] := 2.0;
   DATA[2411,16] := 1.0;
   DATA[2411,17] := 1.0;
   DATA[2411,18] := 1.0;
   DATA[2411,19] := 2.0;
   DATA[2411,20] := 148.808;
   DATA[2411,21] := 155.3448;
   DATA[2411,22] := 1.715824;
   DATA[2411,23] := 859.5104;
   DATA[2411,24] := 2.0;
   DATA[2411,25] := 2.0;
   DATA[2411,26] := 7.874135;
   DATA[2411,27] := 144.4501;
   DATA[2411,28] := 261.5996;
   DATA[2411,29] := 11.95847;
   DATA[2411,30] := 1.724301;
   DATA[2411,31] := 1.281286;
   DATA[2411,32] := 0.7353967;
   DATA[2411,33] := 0.3084265;
   DATA[2411,34] := 2.0;
   DATA[2411,35] := 249.8718;
   DATA[2411,36] := 1.69801;
   DATA[2411,37] := 188.9259;
   DATA[2411,38] := 0.000128152;
   DATA[2411,39] := 1.0;
   DATA[2411,40] := 1.0;
   DATA[2412,0] := 2.619543;
   DATA[2412,1] := 866.3476;
   DATA[2412,2] := 2.0;
   DATA[2412,3] := 2.0;
   DATA[2412,4] := 262.3366;
   DATA[2412,5] := 8.394514;
   DATA[2412,6] := 329.6591;
   DATA[2412,7] := 2.456284;
   DATA[2412,8] := 2.0;
   DATA[2412,9] := 2.0;
   DATA[2412,10] := 2.0;
   DATA[2412,11] := 19.76759;
   DATA[2412,12] := 2.207988;
   DATA[2412,13] := 820.3425;
   DATA[2412,14] := 1.0;
   DATA[2412,15] := 2.0;
   DATA[2412,16] := 1.0;
   DATA[2412,17] := 1.0;
   DATA[2412,18] := 1.0;
   DATA[2412,19] := 2.0;
   DATA[2412,20] := 148.808;
   DATA[2412,21] := 155.3448;
   DATA[2412,22] := 1.715824;
   DATA[2412,23] := 859.8564;
   DATA[2412,24] := 2.0;
   DATA[2412,25] := 2.0;
   DATA[2412,26] := 7.874135;
   DATA[2412,27] := 144.4501;
   DATA[2412,28] := 261.5996;
   DATA[2412,29] := 11.95847;
   DATA[2412,30] := 1.724301;
   DATA[2412,31] := 1.291277;
   DATA[2412,32] := 0.7353967;
   DATA[2412,33] := 0.3084265;
   DATA[2412,34] := 2.0;
   DATA[2412,35] := 250.0;
   DATA[2412,36] := 1.69801;
   DATA[2412,37] := 188.9259;
   DATA[2412,38] := 0.000128152;
   DATA[2412,39] := 1.0;
   DATA[2412,40] := 1.0;
   DATA[2413,0] := 2.614099;
   DATA[2413,1] := 865.9943;
   DATA[2413,2] := 2.0;
   DATA[2413,3] := 2.0;
   DATA[2413,4] := 262.3366;
   DATA[2413,5] := 8.394514;
   DATA[2413,6] := 329.6591;
   DATA[2413,7] := 2.454875;
   DATA[2413,8] := 2.0;
   DATA[2413,9] := 2.0;
   DATA[2413,10] := 2.0;
   DATA[2413,11] := 19.76759;
   DATA[2413,12] := 2.208756;
   DATA[2413,13] := 820.4627;
   DATA[2413,14] := 1.0;
   DATA[2413,15] := 2.0;
   DATA[2413,16] := 1.0;
   DATA[2413,17] := 1.0;
   DATA[2413,18] := 1.0;
   DATA[2413,19] := 2.0;
   DATA[2413,20] := 148.808;
   DATA[2413,21] := 155.3448;
   DATA[2413,22] := 1.715824;
   DATA[2413,23] := 860.2794;
   DATA[2413,24] := 2.0;
   DATA[2413,25] := 2.0;
   DATA[2413,26] := 7.874135;
   DATA[2413,27] := 144.4501;
   DATA[2413,28] := 261.5996;
   DATA[2413,29] := 11.95847;
   DATA[2413,30] := 1.724301;
   DATA[2413,31] := 1.302037;
   DATA[2413,32] := 0.7353967;
   DATA[2413,33] := 0.3084265;
   DATA[2413,34] := 2.0;
   DATA[2413,35] := 250.016;
   DATA[2413,36] := 1.69801;
   DATA[2413,37] := 188.9259;
   DATA[2413,38] := 0.000128152;
   DATA[2413,39] := 1.0;
   DATA[2413,40] := 1.0;
   DATA[2414,0] := 2.60481;
   DATA[2414,1] := 865.9158;
   DATA[2414,2] := 2.0;
   DATA[2414,3] := 2.0;
   DATA[2414,4] := 262.3366;
   DATA[2414,5] := 8.396757;
   DATA[2414,6] := 329.7872;
   DATA[2414,7] := 2.454875;
   DATA[2414,8] := 2.0;
   DATA[2414,9] := 2.0;
   DATA[2414,10] := 2.0;
   DATA[2414,11] := 19.76759;
   DATA[2414,12] := 2.208756;
   DATA[2414,13] := 820.0222;
   DATA[2414,14] := 1.0;
   DATA[2414,15] := 2.0;
   DATA[2414,16] := 1.0;
   DATA[2414,17] := 1.0;
   DATA[2414,18] := 1.0;
   DATA[2414,19] := 2.0;
   DATA[2414,20] := 148.808;
   DATA[2414,21] := 155.3448;
   DATA[2414,22] := 1.717233;
   DATA[2414,23] := 860.4717;
   DATA[2414,24] := 2.0;
   DATA[2414,25] := 2.0;
   DATA[2414,26] := 7.874135;
   DATA[2414,27] := 144.4501;
   DATA[2414,28] := 261.5996;
   DATA[2414,29] := 11.95847;
   DATA[2414,30] := 1.724301;
   DATA[2414,31] := 1.302037;
   DATA[2414,32] := 0.7353967;
   DATA[2414,33] := 0.3084265;
   DATA[2414,34] := 2.0;
   DATA[2414,35] := 250.016;
   DATA[2414,36] := 1.69801;
   DATA[2414,37] := 188.8138;
   DATA[2414,38] := 0.000128152;
   DATA[2414,39] := 1.0;
   DATA[2414,40] := 1.0;
   DATA[2415,0] := 2.579509;
   DATA[2415,1] := 866.1514;
   DATA[2415,2] := 2.0;
   DATA[2415,3] := 2.0;
   DATA[2415,4] := 262.3366;
   DATA[2415,5] := 8.396757;
   DATA[2415,6] := 329.7872;
   DATA[2415,7] := 2.455515;
   DATA[2415,8] := 2.0;
   DATA[2415,9] := 2.0;
   DATA[2415,10] := 2.0;
   DATA[2415,11] := 19.79;
   DATA[2415,12] := 2.209653;
   DATA[2415,13] := 820.5829;
   DATA[2415,14] := 1.0;
   DATA[2415,15] := 2.0;
   DATA[2415,16] := 1.0;
   DATA[2415,17] := 1.0;
   DATA[2415,18] := 1.0;
   DATA[2415,19] := 2.0;
   DATA[2415,20] := 148.808;
   DATA[2415,21] := 155.3448;
   DATA[2415,22] := 1.717361;
   DATA[2415,23] := 860.7024;
   DATA[2415,24] := 2.0;
   DATA[2415,25] := 2.0;
   DATA[2415,26] := 7.874135;
   DATA[2415,27] := 144.5014;
   DATA[2415,28] := 261.5996;
   DATA[2415,29] := 11.95847;
   DATA[2415,30] := 1.726737;
   DATA[2415,31] := 1.302037;
   DATA[2415,32] := 0.7353967;
   DATA[2415,33] := 0.3084265;
   DATA[2415,34] := 2.0;
   DATA[2415,35] := 250.016;
   DATA[2415,36] := 1.69801;
   DATA[2415,37] := 188.8138;
   DATA[2415,38] := 0.000128152;
   DATA[2415,39] := 1.0;
   DATA[2415,40] := 1.0;
   DATA[2416,0] := 2.561573;
   DATA[2416,1] := 866.0729;
   DATA[2416,2] := 2.0;
   DATA[2416,3] := 2.0;
   DATA[2416,4] := 262.3366;
   DATA[2416,5] := 8.396757;
   DATA[2416,6] := 329.7872;
   DATA[2416,7] := 2.456156;
   DATA[2416,8] := 2.0;
   DATA[2416,9] := 2.0;
   DATA[2416,10] := 2.0;
   DATA[2416,11] := 19.83162;
   DATA[2416,12] := 2.209653;
   DATA[2416,13] := 820.4227;
   DATA[2416,14] := 1.0;
   DATA[2416,15] := 2.0;
   DATA[2416,16] := 1.0;
   DATA[2416,17] := 1.0;
   DATA[2416,18] := 1.0;
   DATA[2416,19] := 2.0;
   DATA[2416,20] := 148.808;
   DATA[2416,21] := 155.3448;
   DATA[2416,22] := 1.717361;
   DATA[2416,23] := 860.8947;
   DATA[2416,24] := 2.0;
   DATA[2416,25] := 2.0;
   DATA[2416,26] := 7.874135;
   DATA[2416,27] := 144.527;
   DATA[2416,28] := 261.5996;
   DATA[2416,29] := 11.95847;
   DATA[2416,30] := 1.726737;
   DATA[2416,31] := 1.302037;
   DATA[2416,32] := 0.7353967;
   DATA[2416,33] := 0.3084265;
   DATA[2416,34] := 2.0;
   DATA[2416,35] := 250.1762;
   DATA[2416,36] := 1.890238;
   DATA[2416,37] := 188.8138;
   DATA[2416,38] := 0.000128152;
   DATA[2416,39] := 1.0;
   DATA[2416,40] := 1.0;
   DATA[2417,0] := 2.542036;
   DATA[2417,1] := 866.1906;
   DATA[2417,2] := 2.0;
   DATA[2417,3] := 2.0;
   DATA[2417,4] := 262.3366;
   DATA[2417,5] := 8.396757;
   DATA[2417,6] := 329.7872;
   DATA[2417,7] := 2.456156;
   DATA[2417,8] := 2.0;
   DATA[2417,9] := 2.0;
   DATA[2417,10] := 2.0;
   DATA[2417,11] := 19.84762;
   DATA[2417,12] := 2.209653;
   DATA[2417,13] := 820.7431;
   DATA[2417,14] := 1.0;
   DATA[2417,15] := 2.0;
   DATA[2417,16] := 1.0;
   DATA[2417,17] := 1.0;
   DATA[2417,18] := 1.0;
   DATA[2417,19] := 2.0;
   DATA[2417,20] := 148.808;
   DATA[2417,21] := 155.3448;
   DATA[2417,22] := 1.717361;
   DATA[2417,23] := 860.7024;
   DATA[2417,24] := 2.0;
   DATA[2417,25] := 2.0;
   DATA[2417,26] := 7.874135;
   DATA[2417,27] := 144.527;
   DATA[2417,28] := 261.5996;
   DATA[2417,29] := 11.95847;
   DATA[2417,30] := 1.726737;
   DATA[2417,31] := 1.295888;
   DATA[2417,32] := 0.7353967;
   DATA[2417,33] := 0.3084265;
   DATA[2417,34] := 2.0;
   DATA[2417,35] := 250.1762;
   DATA[2417,36] := 1.826162;
   DATA[2417,37] := 188.8618;
   DATA[2417,38] := 0.000128152;
   DATA[2417,39] := 1.0;
   DATA[2417,40] := 1.0;
   DATA[2418,0] := 2.528264;
   DATA[2418,1] := 866.3083;
   DATA[2418,2] := 2.0;
   DATA[2418,3] := 2.0;
   DATA[2418,4] := 262.3366;
   DATA[2418,5] := 8.396757;
   DATA[2418,6] := 329.7872;
   DATA[2418,7] := 2.456156;
   DATA[2418,8] := 2.0;
   DATA[2418,9] := 2.0;
   DATA[2418,10] := 2.0;
   DATA[2418,11] := 19.84762;
   DATA[2418,12] := 2.209653;
   DATA[2418,13] := 820.3826;
   DATA[2418,14] := 1.0;
   DATA[2418,15] := 2.0;
   DATA[2418,16] := 1.0;
   DATA[2418,17] := 1.0;
   DATA[2418,18] := 1.0;
   DATA[2418,19] := 2.0;
   DATA[2418,20] := 148.808;
   DATA[2418,21] := 155.2935;
   DATA[2418,22] := 1.718771;
   DATA[2418,23] := 861.2407;
   DATA[2418,24] := 2.0;
   DATA[2418,25] := 2.0;
   DATA[2418,26] := 7.874135;
   DATA[2418,27] := 144.527;
   DATA[2418,28] := 261.5996;
   DATA[2418,29] := 11.95847;
   DATA[2418,30] := 1.728659;
   DATA[2418,31] := 1.283079;
   DATA[2418,32] := 0.7353967;
   DATA[2418,33] := 0.3084265;
   DATA[2418,34] := 2.0;
   DATA[2418,35] := 250.1762;
   DATA[2418,36] := 1.762086;
   DATA[2418,37] := 189.006;
   DATA[2418,38] := 0.000128152;
   DATA[2418,39] := 1.0;
   DATA[2418,40] := 1.0;
   DATA[2419,0] := 2.504244;
   DATA[2419,1] := 866.5439;
   DATA[2419,2] := 2.0;
   DATA[2419,3] := 2.0;
   DATA[2419,4] := 262.3366;
   DATA[2419,5] := 8.396757;
   DATA[2419,6] := 329.7872;
   DATA[2419,7] := 2.456156;
   DATA[2419,8] := 2.0;
   DATA[2419,9] := 2.0;
   DATA[2419,10] := 2.0;
   DATA[2419,11] := 19.84762;
   DATA[2419,12] := 2.209653;
   DATA[2419,13] := 820.8232;
   DATA[2419,14] := 1.0;
   DATA[2419,15] := 2.0;
   DATA[2419,16] := 1.0;
   DATA[2419,17] := 1.0;
   DATA[2419,18] := 1.0;
   DATA[2419,19] := 2.0;
   DATA[2419,20] := 148.808;
   DATA[2419,21] := 155.2935;
   DATA[2419,22] := 1.719156;
   DATA[2419,23] := 861.7021;
   DATA[2419,24] := 2.0;
   DATA[2419,25] := 2.0;
   DATA[2419,26] := 7.874135;
   DATA[2419,27] := 144.527;
   DATA[2419,28] := 261.5996;
   DATA[2419,29] := 11.95847;
   DATA[2419,30] := 1.728659;
   DATA[2419,31] := 1.282183;
   DATA[2419,32] := 0.7353967;
   DATA[2419,33] := 0.3084265;
   DATA[2419,34] := 2.0;
   DATA[2419,35] := 250.1762;
   DATA[2419,36] := 1.665972;
   DATA[2419,37] := 189.0381;
   DATA[2419,38] := 0.000128152;
   DATA[2419,39] := 1.0;
   DATA[2419,40] := 1.0;
   DATA[2420,0] := 2.489191;
   DATA[2420,1] := 866.4654;
   DATA[2420,2] := 2.0;
   DATA[2420,3] := 2.0;
   DATA[2420,4] := 262.3366;
   DATA[2420,5] := 8.396757;
   DATA[2420,6] := 329.7872;
   DATA[2420,7] := 2.456156;
   DATA[2420,8] := 2.0;
   DATA[2420,9] := 2.0;
   DATA[2420,10] := 2.0;
   DATA[2420,11] := 19.77079;
   DATA[2420,12] := 2.208756;
   DATA[2420,13] := 820.6229;
   DATA[2420,14] := 1.0;
   DATA[2420,15] := 2.0;
   DATA[2420,16] := 1.0;
   DATA[2420,17] := 1.0;
   DATA[2420,18] := 1.0;
   DATA[2420,19] := 2.0;
   DATA[2420,20] := 148.808;
   DATA[2420,21] := 155.2935;
   DATA[2420,22] := 1.719284;
   DATA[2420,23] := 861.6637;
   DATA[2420,24] := 2.0;
   DATA[2420,25] := 2.0;
   DATA[2420,26] := 7.874135;
   DATA[2420,27] := 144.527;
   DATA[2420,28] := 261.5996;
   DATA[2420,29] := 11.95847;
   DATA[2420,30] := 1.728916;
   DATA[2420,31] := 1.272576;
   DATA[2420,32] := 0.7353967;
   DATA[2420,33] := 0.306761;
   DATA[2420,34] := 2.0;
   DATA[2420,35] := 250.2403;
   DATA[2420,36] := 1.665972;
   DATA[2420,37] := 189.1182;
   DATA[2420,38] := 0.000128152;
   DATA[2420,39] := 1.0;
   DATA[2420,40] := 1.0;
   DATA[2421,0] := 2.471255;
   DATA[2421,1] := 866.5831;
   DATA[2421,2] := 2.0;
   DATA[2421,3] := 2.0;
   DATA[2421,4] := 262.3366;
   DATA[2421,5] := 8.395155;
   DATA[2421,6] := 329.7872;
   DATA[2421,7] := 2.456156;
   DATA[2421,8] := 2.0;
   DATA[2421,9] := 2.0;
   DATA[2421,10] := 2.0;
   DATA[2421,11] := 19.72598;
   DATA[2421,12] := 2.208116;
   DATA[2421,13] := 820.9434;
   DATA[2421,14] := 1.0;
   DATA[2421,15] := 2.0;
   DATA[2421,16] := 1.0;
   DATA[2421,17] := 1.0;
   DATA[2421,18] := 1.0;
   DATA[2421,19] := 2.0;
   DATA[2421,20] := 148.808;
   DATA[2421,21] := 155.2935;
   DATA[2421,22] := 1.720693;
   DATA[2421,23] := 862.202;
   DATA[2421,24] := 2.0;
   DATA[2421,25] := 2.0;
   DATA[2421,26] := 7.874135;
   DATA[2421,27] := 144.527;
   DATA[2421,28] := 261.5996;
   DATA[2421,29] := 11.95847;
   DATA[2421,30] := 1.728916;
   DATA[2421,31] := 1.272064;
   DATA[2421,32] := 0.7353967;
   DATA[2421,33] := 0.306761;
   DATA[2421,34] := 2.0;
   DATA[2421,35] := 250.2724;
   DATA[2421,36] := 1.665972;
   DATA[2421,37] := 189.1182;
   DATA[2421,38] := 0.000128152;
   DATA[2421,39] := 1.0;
   DATA[2421,40] := 1.0;
   DATA[2422,0] := 2.456843;
   DATA[2422,1] := 866.5046;
   DATA[2422,2] := 2.0;
   DATA[2422,3] := 2.0;
   DATA[2422,4] := 262.3366;
   DATA[2422,5] := 8.395155;
   DATA[2422,6] := 329.7872;
   DATA[2422,7] := 2.456156;
   DATA[2422,8] := 2.0;
   DATA[2422,9] := 2.0;
   DATA[2422,10] := 2.0;
   DATA[2422,11] := 19.72598;
   DATA[2422,12] := 2.207091;
   DATA[2422,13] := 820.7831;
   DATA[2422,14] := 1.0;
   DATA[2422,15] := 2.0;
   DATA[2422,16] := 1.0;
   DATA[2422,17] := 1.0;
   DATA[2422,18] := 1.0;
   DATA[2422,19] := 2.0;
   DATA[2422,20] := 148.808;
   DATA[2422,21] := 155.2935;
   DATA[2422,22] := 1.722872;
   DATA[2422,23] := 862.6249;
   DATA[2422,24] := 2.0;
   DATA[2422,25] := 2.0;
   DATA[2422,26] := 7.874135;
   DATA[2422,27] := 144.527;
   DATA[2422,28] := 261.5996;
   DATA[2422,29] := 11.95847;
   DATA[2422,30] := 1.728916;
   DATA[2422,31] := 1.288843;
   DATA[2422,32] := 0.7353967;
   DATA[2422,33] := 0.306761;
   DATA[2422,34] := 2.0;
   DATA[2422,35] := 250.2724;
   DATA[2422,36] := 1.665972;
   DATA[2422,37] := 189.1182;
   DATA[2422,38] := 0.000128152;
   DATA[2422,39] := 1.0;
   DATA[2422,40] := 1.0;
   DATA[2423,0] := 2.456843;
   DATA[2423,1] := 866.5046;
   DATA[2423,2] := 2.0;
   DATA[2423,3] := 2.0;
   DATA[2423,4] := 262.3366;
   DATA[2423,5] := 8.395155;
   DATA[2423,6] := 329.7872;
   DATA[2423,7] := 2.456156;
   DATA[2423,8] := 2.0;
   DATA[2423,9] := 2.0;
   DATA[2423,10] := 2.0;
   DATA[2423,11] := 19.72598;
   DATA[2423,12] := 2.207091;
   DATA[2423,13] := 820.7831;
   DATA[2423,14] := 1.0;
   DATA[2423,15] := 2.0;
   DATA[2423,16] := 1.0;
   DATA[2423,17] := 1.0;
   DATA[2423,18] := 1.0;
   DATA[2423,19] := 2.0;
   DATA[2423,20] := 148.808;
   DATA[2423,21] := 155.2935;
   DATA[2423,22] := 1.722872;
   DATA[2423,23] := 862.6249;
   DATA[2423,24] := 2.0;
   DATA[2423,25] := 2.0;
   DATA[2423,26] := 7.874135;
   DATA[2423,27] := 144.527;
   DATA[2423,28] := 261.5996;
   DATA[2423,29] := 11.95847;
   DATA[2423,30] := 1.728916;
   DATA[2423,31] := 1.288843;
   DATA[2423,32] := 0.7353967;
   DATA[2423,33] := 0.306761;
   DATA[2423,34] := 2.0;
   DATA[2423,35] := 250.2724;
   DATA[2423,36] := 1.665972;
   DATA[2423,37] := 189.1182;
   DATA[2423,38] := 0.000128152;
   DATA[2423,39] := 1.0;
   DATA[2423,40] := 1.0;
   DATA[2424,0] := 2.436345;
   DATA[2424,1] := 866.7794;
   DATA[2424,2] := 2.0;
   DATA[2424,3] := 2.0;
   DATA[2424,4] := 262.3366;
   DATA[2424,5] := 8.395155;
   DATA[2424,6] := 329.7872;
   DATA[2424,7] := 2.453849;
   DATA[2424,8] := 2.0;
   DATA[2424,9] := 2.0;
   DATA[2424,10] := 2.0;
   DATA[2424,11] := 19.70357;
   DATA[2424,12] := 2.20581;
   DATA[2424,13] := 821.0235;
   DATA[2424,14] := 1.0;
   DATA[2424,15] := 2.0;
   DATA[2424,16] := 1.0;
   DATA[2424,17] := 1.0;
   DATA[2424,18] := 1.0;
   DATA[2424,19] := 2.0;
   DATA[2424,20] := 148.808;
   DATA[2424,21] := 155.2935;
   DATA[2424,22] := 1.722872;
   DATA[2424,23] := 862.6634;
   DATA[2424,24] := 2.0;
   DATA[2424,25] := 2.0;
   DATA[2424,26] := 7.874135;
   DATA[2424,27] := 144.527;
   DATA[2424,28] := 261.5996;
   DATA[2424,29] := 11.95847;
   DATA[2424,30] := 1.728916;
   DATA[2424,31] := 1.291789;
   DATA[2424,32] := 0.7353967;
   DATA[2424,33] := 0.306761;
   DATA[2424,34] := 2.0;
   DATA[2424,35] := 250.2724;
   DATA[2424,36] := 1.665972;
   DATA[2424,37] := 189.1182;
   DATA[2424,38] := 0.000128152;
   DATA[2424,39] := 1.0;
   DATA[2424,40] := 1.0;
   DATA[2425,0] := 2.424815;
   DATA[2425,1] := 866.7009;
   DATA[2425,2] := 2.0;
   DATA[2425,3] := 2.0;
   DATA[2425,4] := 262.3366;
   DATA[2425,5] := 8.395155;
   DATA[2425,6] := 329.7872;
   DATA[2425,7] := 2.453721;
   DATA[2425,8] := 2.0;
   DATA[2425,9] := 2.0;
   DATA[2425,10] := 2.0;
   DATA[2425,11] := 19.67476;
   DATA[2425,12] := 2.205426;
   DATA[2425,13] := 821.384;
   DATA[2425,14] := 1.0;
   DATA[2425,15] := 2.0;
   DATA[2425,16] := 1.0;
   DATA[2425,17] := 1.0;
   DATA[2425,18] := 1.0;
   DATA[2425,19] := 2.0;
   DATA[2425,20] := 148.808;
   DATA[2425,21] := 155.3448;
   DATA[2425,22] := 1.722872;
   DATA[2425,23] := 863.2402;
   DATA[2425,24] := 2.0;
   DATA[2425,25] := 2.0;
   DATA[2425,26] := 7.874135;
   DATA[2425,27] := 144.527;
   DATA[2425,28] := 261.5996;
   DATA[2425,29] := 11.95847;
   DATA[2425,30] := 1.726609;
   DATA[2425,31] := 1.291277;
   DATA[2425,32] := 0.7353967;
   DATA[2425,33] := 0.306761;
   DATA[2425,34] := 2.0;
   DATA[2425,35] := 250.2724;
   DATA[2425,36] := 1.665972;
   DATA[2425,37] := 189.1182;
   DATA[2425,38] := 0.000128152;
   DATA[2425,39] := 1.0;
   DATA[2425,40] := 1.0;
   DATA[2426,0] := 2.423213;
   DATA[2426,1] := 866.9364;
   DATA[2426,2] := 2.0;
   DATA[2426,3] := 2.0;
   DATA[2426,4] := 262.3366;
   DATA[2426,5] := 8.395155;
   DATA[2426,6] := 329.7872;
   DATA[2426,7] := 2.453721;
   DATA[2426,8] := 2.0;
   DATA[2426,9] := 2.0;
   DATA[2426,10] := 2.0;
   DATA[2426,11] := 19.70037;
   DATA[2426,12] := 2.205426;
   DATA[2426,13] := 821.4641;
   DATA[2426,14] := 1.0;
   DATA[2426,15] := 2.0;
   DATA[2426,16] := 1.0;
   DATA[2426,17] := 1.0;
   DATA[2426,18] := 1.0;
   DATA[2426,19] := 2.0;
   DATA[2426,20] := 148.808;
   DATA[2426,21] := 155.3448;
   DATA[2426,22] := 1.720565;
   DATA[2426,23] := 863.1633;
   DATA[2426,24] := 2.0;
   DATA[2426,25] := 2.0;
   DATA[2426,26] := 7.874135;
   DATA[2426,27] := 144.527;
   DATA[2426,28] := 261.5996;
   DATA[2426,29] := 11.95847;
   DATA[2426,30] := 1.726609;
   DATA[2426,31] := 1.286922;
   DATA[2426,32] := 0.7353967;
   DATA[2426,33] := 0.306761;
   DATA[2426,34] := 2.0;
   DATA[2426,35] := 250.2724;
   DATA[2426,36] := 1.665972;
   DATA[2426,37] := 189.1182;
   DATA[2426,38] := 0.000128152;
   DATA[2426,39] := 1.0;
   DATA[2426,40] := 1.0;
   DATA[2427,0] := 2.425135;
   DATA[2427,1] := 867.0934;
   DATA[2427,2] := 2.0;
   DATA[2427,3] := 2.0;
   DATA[2427,4] := 262.3366;
   DATA[2427,5] := 8.395155;
   DATA[2427,6] := 329.7872;
   DATA[2427,7] := 2.45308;
   DATA[2427,8] := 2.0;
   DATA[2427,9] := 2.0;
   DATA[2427,10] := 2.0;
   DATA[2427,11] := 19.72277;
   DATA[2427,12] := 2.205426;
   DATA[2427,13] := 821.6643;
   DATA[2427,14] := 1.0;
   DATA[2427,15] := 2.0;
   DATA[2427,16] := 1.0;
   DATA[2427,17] := 1.0;
   DATA[2427,18] := 1.0;
   DATA[2427,19] := 2.0;
   DATA[2427,20] := 148.808;
   DATA[2427,21] := 155.3448;
   DATA[2427,22] := 1.720053;
   DATA[2427,23] := 863.3555;
   DATA[2427,24] := 2.0;
   DATA[2427,25] := 2.0;
   DATA[2427,26] := 7.874135;
   DATA[2427,27] := 144.527;
   DATA[2427,28] := 261.5996;
   DATA[2427,29] := 11.95847;
   DATA[2427,30] := 1.726609;
   DATA[2427,31] := 1.287691;
   DATA[2427,32] := 0.7353967;
   DATA[2427,33] := 0.30785;
   DATA[2427,34] := 2.0;
   DATA[2427,35] := 250.2724;
   DATA[2427,36] := 1.762086;
   DATA[2427,37] := 189.1182;
   DATA[2427,38] := 0.000128152;
   DATA[2427,39] := 1.0;
   DATA[2427,40] := 1.0;
   DATA[2428,0] := 2.461647;
   DATA[2428,1] := 867.2897;
   DATA[2428,2] := 2.0;
   DATA[2428,3] := 2.0;
   DATA[2428,4] := 262.3366;
   DATA[2428,5] := 8.395155;
   DATA[2428,6] := 329.7872;
   DATA[2428,7] := 2.451927;
   DATA[2428,8] := 2.0;
   DATA[2428,9] := 2.0;
   DATA[2428,10] := 2.0;
   DATA[2428,11] := 19.72277;
   DATA[2428,12] := 2.205426;
   DATA[2428,13] := 821.8646;
   DATA[2428,14] := 1.0;
   DATA[2428,15] := 2.0;
   DATA[2428,16] := 1.0;
   DATA[2428,17] := 1.0;
   DATA[2428,18] := 1.0;
   DATA[2428,19] := 2.0;
   DATA[2428,20] := 148.808;
   DATA[2428,21] := 155.3448;
   DATA[2428,22] := 1.720053;
   DATA[2428,23] := 863.1633;
   DATA[2428,24] := 2.0;
   DATA[2428,25] := 2.0;
   DATA[2428,26] := 7.874135;
   DATA[2428,27] := 144.527;
   DATA[2428,28] := 261.5996;
   DATA[2428,29] := 11.95847;
   DATA[2428,30] := 1.726609;
   DATA[2428,31] := 1.287691;
   DATA[2428,32] := 0.7353967;
   DATA[2428,33] := 0.30785;
   DATA[2428,34] := 2.0;
   DATA[2428,35] := 250.2724;
   DATA[2428,36] := 1.762086;
   DATA[2428,37] := 189.1182;
   DATA[2428,38] := 0.000128152;
   DATA[2428,39] := 1.0;
   DATA[2428,40] := 1.0;
   DATA[2429,0] := 2.506806;
   DATA[2429,1] := 867.2897;
   DATA[2429,2] := 2.0;
   DATA[2429,3] := 2.0;
   DATA[2429,4] := 262.3366;
   DATA[2429,5] := 8.395155;
   DATA[2429,6] := 329.7872;
   DATA[2429,7] := 2.451671;
   DATA[2429,8] := 2.0;
   DATA[2429,9] := 2.0;
   DATA[2429,10] := 2.0;
   DATA[2429,11] := 19.72277;
   DATA[2429,12] := 2.205426;
   DATA[2429,13] := 821.9447;
   DATA[2429,14] := 1.0;
   DATA[2429,15] := 2.0;
   DATA[2429,16] := 1.0;
   DATA[2429,17] := 1.0;
   DATA[2429,18] := 1.0;
   DATA[2429,19] := 2.0;
   DATA[2429,20] := 148.808;
   DATA[2429,21] := 155.3448;
   DATA[2429,22] := 1.720053;
   DATA[2429,23] := 863.394;
   DATA[2429,24] := 2.0;
   DATA[2429,25] := 2.0;
   DATA[2429,26] := 7.874135;
   DATA[2429,27] := 144.527;
   DATA[2429,28] := 261.5996;
   DATA[2429,29] := 11.95847;
   DATA[2429,30] := 1.726609;
   DATA[2429,31] := 1.302677;
   DATA[2429,32] := 0.7353967;
   DATA[2429,33] := 0.30785;
   DATA[2429,34] := 2.0;
   DATA[2429,35] := 250.2724;
   DATA[2429,36] := 1.762086;
   DATA[2429,37] := 189.1182;
   DATA[2429,38] := 0.000128152;
   DATA[2429,39] := 1.0;
   DATA[2429,40] := 1.0;
   DATA[2430,0] := 2.550043;
   DATA[2430,1] := 867.1719;
   DATA[2430,2] := 2.0;
   DATA[2430,3] := 2.0;
   DATA[2430,4] := 262.3366;
   DATA[2430,5] := 8.395155;
   DATA[2430,6] := 329.7872;
   DATA[2430,7] := 2.450774;
   DATA[2430,8] := 2.0;
   DATA[2430,9] := 2.0;
   DATA[2430,10] := 2.0;
   DATA[2430,11] := 19.72277;
   DATA[2430,12] := 2.205426;
   DATA[2430,13] := 822.1851;
   DATA[2430,14] := 1.0;
   DATA[2430,15] := 2.0;
   DATA[2430,16] := 1.0;
   DATA[2430,17] := 1.0;
   DATA[2430,18] := 1.0;
   DATA[2430,19] := 2.0;
   DATA[2430,20] := 148.808;
   DATA[2430,21] := 155.3448;
   DATA[2430,22] := 1.720053;
   DATA[2430,23] := 863.2402;
   DATA[2430,24] := 2.0;
   DATA[2430,25] := 2.0;
   DATA[2430,26] := 7.874135;
   DATA[2430,27] := 144.527;
   DATA[2430,28] := 261.5996;
   DATA[2430,29] := 11.95847;
   DATA[2430,30] := 1.726609;
   DATA[2430,31] := 1.307288;
   DATA[2430,32] := 0.7353967;
   DATA[2430,33] := 0.30785;
   DATA[2430,34] := 2.0;
   DATA[2430,35] := 250.2724;
   DATA[2430,36] := 1.762086;
   DATA[2430,37] := 189.1182;
   DATA[2430,38] := 0.000128152;
   DATA[2430,39] := 1.0;
   DATA[2430,40] := 1.0;
   DATA[2431,0] := 2.572783;
   DATA[2431,1] := 866.9756;
   DATA[2431,2] := 2.0;
   DATA[2431,3] := 2.0;
   DATA[2431,4] := 262.3366;
   DATA[2431,5] := 8.395155;
   DATA[2431,6] := 329.7872;
   DATA[2431,7] := 2.450389;
   DATA[2431,8] := 2.0;
   DATA[2431,9] := 2.0;
   DATA[2431,10] := 2.0;
   DATA[2431,11] := 19.75799;
   DATA[2431,12] := 2.207347;
   DATA[2431,13] := 822.3453;
   DATA[2431,14] := 1.0;
   DATA[2431,15] := 2.0;
   DATA[2431,16] := 1.0;
   DATA[2431,17] := 1.0;
   DATA[2431,18] := 1.0;
   DATA[2431,19] := 2.0;
   DATA[2431,20] := 148.808;
   DATA[2431,21] := 155.3448;
   DATA[2431,22] := 1.720053;
   DATA[2431,23] := 863.2402;
   DATA[2431,24] := 2.0;
   DATA[2431,25] := 2.0;
   DATA[2431,26] := 7.874135;
   DATA[2431,27] := 144.527;
   DATA[2431,28] := 261.5996;
   DATA[2431,29] := 11.95847;
   DATA[2431,30] := 1.726609;
   DATA[2431,31] := 1.307288;
   DATA[2431,32] := 0.7353967;
   DATA[2431,33] := 0.3072094;
   DATA[2431,34] := 2.0;
   DATA[2431,35] := 250.2724;
   DATA[2431,36] := 1.762086;
   DATA[2431,37] := 189.1182;
   DATA[2431,38] := 0.000128152;
   DATA[2431,39] := 1.0;
   DATA[2431,40] := 1.0;
   DATA[2432,0] := 2.625308;
   DATA[2432,1] := 867.0542;
   DATA[2432,2] := 2.0;
   DATA[2432,3] := 2.0;
   DATA[2432,4] := 262.3366;
   DATA[2432,5] := 8.395155;
   DATA[2432,6] := 329.7872;
   DATA[2432,7] := 2.451286;
   DATA[2432,8] := 2.0;
   DATA[2432,9] := 2.0;
   DATA[2432,10] := 2.0;
   DATA[2432,11] := 19.77399;
   DATA[2432,12] := 2.208756;
   DATA[2432,13] := 822.2651;
   DATA[2432,14] := 1.0;
   DATA[2432,15] := 2.0;
   DATA[2432,16] := 1.0;
   DATA[2432,17] := 1.0;
   DATA[2432,18] := 1.0;
   DATA[2432,19] := 2.0;
   DATA[2432,20] := 148.808;
   DATA[2432,21] := 155.3448;
   DATA[2432,22] := 1.717233;
   DATA[2432,23] := 863.394;
   DATA[2432,24] := 2.0;
   DATA[2432,25] := 2.0;
   DATA[2432,26] := 7.874135;
   DATA[2432,27] := 144.4501;
   DATA[2432,28] := 261.5996;
   DATA[2432,29] := 11.95847;
   DATA[2432,30] := 1.726609;
   DATA[2432,31] := 1.308057;
   DATA[2432,32] := 0.7353967;
   DATA[2432,33] := 0.3063127;
   DATA[2432,34] := 2.0;
   DATA[2432,35] := 250.2724;
   DATA[2432,36] := 1.665972;
   DATA[2432,37] := 189.1182;
   DATA[2432,38] := 0.000128152;
   DATA[2432,39] := 1.0;
   DATA[2432,40] := 1.0;
   DATA[2433,0] := 2.641322;
   DATA[2433,1] := 867.1327;
   DATA[2433,2] := 2.0;
   DATA[2433,3] := 2.0;
   DATA[2433,4] := 262.3366;
   DATA[2433,5] := 8.395155;
   DATA[2433,6] := 329.7872;
   DATA[2433,7] := 2.451927;
   DATA[2433,8] := 2.0;
   DATA[2433,9] := 2.0;
   DATA[2433,10] := 2.0;
   DATA[2433,11] := 19.77399;
   DATA[2433,12] := 2.208756;
   DATA[2433,13] := 822.2651;
   DATA[2433,14] := 1.0;
   DATA[2433,15] := 2.0;
   DATA[2433,16] := 1.0;
   DATA[2433,17] := 1.0;
   DATA[2433,18] := 1.0;
   DATA[2433,19] := 2.0;
   DATA[2433,20] := 148.808;
   DATA[2433,21] := 155.3448;
   DATA[2433,22] := 1.717233;
   DATA[2433,23] := 863.394;
   DATA[2433,24] := 2.0;
   DATA[2433,25] := 2.0;
   DATA[2433,26] := 7.874135;
   DATA[2433,27] := 144.3732;
   DATA[2433,28] := 261.5996;
   DATA[2433,29] := 11.95847;
   DATA[2433,30] := 1.726609;
   DATA[2433,31] := 1.294351;
   DATA[2433,32] := 0.7353967;
   DATA[2433,33] := 0.3063127;
   DATA[2433,34] := 2.0;
   DATA[2433,35] := 250.3365;
   DATA[2433,36] := 1.665972;
   DATA[2433,37] := 189.1182;
   DATA[2433,38] := 0.000128152;
   DATA[2433,39] := 1.0;
   DATA[2433,40] := 1.0;
   DATA[2434,0] := 2.657016;
   DATA[2434,1] := 867.3682;
   DATA[2434,2] := 2.0;
   DATA[2434,3] := 2.0;
   DATA[2434,4] := 262.3366;
   DATA[2434,5] := 8.395155;
   DATA[2434,6] := 329.7872;
   DATA[2434,7] := 2.451927;
   DATA[2434,8] := 2.0;
   DATA[2434,9] := 2.0;
   DATA[2434,10] := 2.0;
   DATA[2434,11] := 19.68436;
   DATA[2434,12] := 2.208756;
   DATA[2434,13] := 822.4654;
   DATA[2434,14] := 1.0;
   DATA[2434,15] := 2.0;
   DATA[2434,16] := 1.0;
   DATA[2434,17] := 1.0;
   DATA[2434,18] := 1.0;
   DATA[2434,19] := 2.0;
   DATA[2434,20] := 148.808;
   DATA[2434,21] := 155.3448;
   DATA[2434,22] := 1.717233;
   DATA[2434,23] := 863.1633;
   DATA[2434,24] := 2.0;
   DATA[2434,25] := 2.0;
   DATA[2434,26] := 7.874135;
   DATA[2434,27] := 144.3732;
   DATA[2434,28] := 261.5996;
   DATA[2434,29] := 11.95847;
   DATA[2434,30] := 1.726609;
   DATA[2434,31] := 1.292046;
   DATA[2434,32] := 0.7353967;
   DATA[2434,33] := 0.3063127;
   DATA[2434,34] := 2.0;
   DATA[2434,35] := 250.3365;
   DATA[2434,36] := 1.665972;
   DATA[2434,37] := 189.1182;
   DATA[2434,38] := 0.000128152;
   DATA[2434,39] := 1.0;
   DATA[2434,40] := 1.0;
   DATA[2435,0] := 2.657016;
   DATA[2435,1] := 867.5645;
   DATA[2435,2] := 2.0;
   DATA[2435,3] := 2.0;
   DATA[2435,4] := 262.3366;
   DATA[2435,5] := 8.395155;
   DATA[2435,6] := 329.7872;
   DATA[2435,7] := 2.451927;
   DATA[2435,8] := 2.0;
   DATA[2435,9] := 2.0;
   DATA[2435,10] := 2.0;
   DATA[2435,11] := 19.68436;
   DATA[2435,12] := 2.208756;
   DATA[2435,13] := 822.6256;
   DATA[2435,14] := 1.0;
   DATA[2435,15] := 2.0;
   DATA[2435,16] := 1.0;
   DATA[2435,17] := 1.0;
   DATA[2435,18] := 1.0;
   DATA[2435,19] := 2.0;
   DATA[2435,20] := 148.808;
   DATA[2435,21] := 155.3448;
   DATA[2435,22] := 1.715567;
   DATA[2435,23] := 863.2402;
   DATA[2435,24] := 2.0;
   DATA[2435,25] := 2.0;
   DATA[2435,26] := 7.874135;
   DATA[2435,27] := 144.3732;
   DATA[2435,28] := 261.5996;
   DATA[2435,29] := 11.95847;
   DATA[2435,30] := 1.726609;
   DATA[2435,31] := 1.283079;
   DATA[2435,32] := 0.7353967;
   DATA[2435,33] := 0.3074656;
   DATA[2435,34] := 2.0;
   DATA[2435,35] := 250.3365;
   DATA[2435,36] := 1.665972;
   DATA[2435,37] := 189.1182;
   DATA[2435,38] := 0.000128152;
   DATA[2435,39] := 1.0;
   DATA[2435,40] := 1.0;
   DATA[2436,0] := 2.631393;
   DATA[2436,1] := 867.0934;
   DATA[2436,2] := 2.0;
   DATA[2436,3] := 2.0;
   DATA[2436,4] := 262.3366;
   DATA[2436,5] := 8.395155;
   DATA[2436,6] := 329.7872;
   DATA[2436,7] := 2.451927;
   DATA[2436,8] := 2.0;
   DATA[2436,9] := 2.0;
   DATA[2436,10] := 2.0;
   DATA[2436,11] := 19.75799;
   DATA[2436,12] := 2.208756;
   DATA[2436,13] := 822.5455;
   DATA[2436,14] := 1.0;
   DATA[2436,15] := 2.0;
   DATA[2436,16] := 1.0;
   DATA[2436,17] := 1.0;
   DATA[2436,18] := 1.0;
   DATA[2436,19] := 2.0;
   DATA[2436,20] := 148.808;
   DATA[2436,21] := 155.3448;
   DATA[2436,22] := 1.715567;
   DATA[2436,23] := 862.7403;
   DATA[2436,24] := 2.0;
   DATA[2436,25] := 2.0;
   DATA[2436,26] := 7.874135;
   DATA[2436,27] := 144.3732;
   DATA[2436,28] := 261.5996;
   DATA[2436,29] := 11.95847;
   DATA[2436,30] := 1.726609;
   DATA[2436,31] := 1.281542;
   DATA[2436,32] := 0.7353967;
   DATA[2436,33] := 0.3075297;
   DATA[2436,34] := 2.0;
   DATA[2436,35] := 250.016;
   DATA[2436,36] := 1.746067;
   DATA[2436,37] := 188.8939;
   DATA[2436,38] := 0.000128152;
   DATA[2436,39] := 1.0;
   DATA[2436,40] := 1.0;
   DATA[2437,0] := 2.623387;
   DATA[2437,1] := 867.486;
   DATA[2437,2] := 2.0;
   DATA[2437,3] := 2.0;
   DATA[2437,4] := 262.3366;
   DATA[2437,5] := 8.395155;
   DATA[2437,6] := 329.7872;
   DATA[2437,7] := 2.453337;
   DATA[2437,8] := 2.0;
   DATA[2437,9] := 2.0;
   DATA[2437,10] := 2.0;
   DATA[2437,11] := 19.7836;
   DATA[2437,12] := 2.207603;
   DATA[2437,13] := 822.7458;
   DATA[2437,14] := 1.0;
   DATA[2437,15] := 2.0;
   DATA[2437,16] := 1.0;
   DATA[2437,17] := 1.0;
   DATA[2437,18] := 1.0;
   DATA[2437,19] := 2.0;
   DATA[2437,20] := 148.808;
   DATA[2437,21] := 155.3448;
   DATA[2437,22] := 1.715567;
   DATA[2437,23] := 862.8172;
   DATA[2437,24] := 2.0;
   DATA[2437,25] := 2.0;
   DATA[2437,26] := 7.874135;
   DATA[2437,27] := 144.3732;
   DATA[2437,28] := 261.5996;
   DATA[2437,29] := 11.95847;
   DATA[2437,30] := 1.726609;
   DATA[2437,31] := 1.282951;
   DATA[2437,32] := 0.7353967;
   DATA[2437,33] := 0.30785;
   DATA[2437,34] := 2.0;
   DATA[2437,35] := 250.016;
   DATA[2437,36] := 1.746067;
   DATA[2437,37] := 188.8939;
   DATA[2437,38] := 0.000128152;
   DATA[2437,39] := 1.0;
   DATA[2437,40] := 1.0;
   DATA[2438,0] := 2.617942;
   DATA[2438,1] := 867.486;
   DATA[2438,2] := 2.0;
   DATA[2438,3] := 2.0;
   DATA[2438,4] := 262.3366;
   DATA[2438,5] := 8.395155;
   DATA[2438,6] := 329.7872;
   DATA[2438,7] := 2.453337;
   DATA[2438,8] := 2.0;
   DATA[2438,9] := 2.0;
   DATA[2438,10] := 2.0;
   DATA[2438,11] := 19.7836;
   DATA[2438,12] := 2.206322;
   DATA[2438,13] := 822.6657;
   DATA[2438,14] := 1.0;
   DATA[2438,15] := 2.0;
   DATA[2438,16] := 1.0;
   DATA[2438,17] := 1.0;
   DATA[2438,18] := 1.0;
   DATA[2438,19] := 2.0;
   DATA[2438,20] := 148.808;
   DATA[2438,21] := 155.3448;
   DATA[2438,22] := 1.713645;
   DATA[2438,23] := 862.5865;
   DATA[2438,24] := 2.0;
   DATA[2438,25] := 2.0;
   DATA[2438,26] := 7.874135;
   DATA[2438,27] := 144.3732;
   DATA[2438,28] := 261.5996;
   DATA[2438,29] := 11.95847;
   DATA[2438,30] := 1.726609;
   DATA[2438,31] := 1.285129;
   DATA[2438,32] := 0.7353967;
   DATA[2438,33] := 0.3081062;
   DATA[2438,34] := 2.0;
   DATA[2438,35] := 250.016;
   DATA[2438,36] := 1.746067;
   DATA[2438,37] := 188.8939;
   DATA[2438,38] := 0.000128152;
   DATA[2438,39] := 1.0;
   DATA[2438,40] := 1.0;
   DATA[2439,0] := 2.605131;
   DATA[2439,1] := 867.2897;
   DATA[2439,2] := 2.0;
   DATA[2439,3] := 2.0;
   DATA[2439,4] := 262.3366;
   DATA[2439,5] := 8.395155;
   DATA[2439,6] := 329.7872;
   DATA[2439,7] := 2.453337;
   DATA[2439,8] := 2.0;
   DATA[2439,9] := 2.0;
   DATA[2439,10] := 2.0;
   DATA[2439,11] := 19.69396;
   DATA[2439,12] := 2.206322;
   DATA[2439,13] := 822.2651;
   DATA[2439,14] := 1.0;
   DATA[2439,15] := 2.0;
   DATA[2439,16] := 1.0;
   DATA[2439,17] := 1.0;
   DATA[2439,18] := 1.0;
   DATA[2439,19] := 2.0;
   DATA[2439,20] := 148.808;
   DATA[2439,21] := 155.3448;
   DATA[2439,22] := 1.713389;
   DATA[2439,23] := 862.2789;
   DATA[2439,24] := 2.0;
   DATA[2439,25] := 2.0;
   DATA[2439,26] := 7.874135;
   DATA[2439,27] := 144.3732;
   DATA[2439,28] := 261.5996;
   DATA[2439,29] := 11.95847;
   DATA[2439,30] := 1.726609;
   DATA[2439,31] := 1.288075;
   DATA[2439,32] := 0.7353967;
   DATA[2439,33] := 0.3081062;
   DATA[2439,34] := 2.0;
   DATA[2439,35] := 250.016;
   DATA[2439,36] := 1.585878;
   DATA[2439,37] := 188.8939;
   DATA[2439,38] := 0.000128152;
   DATA[2439,39] := 1.0;
   DATA[2439,40] := 1.0;
   DATA[2440,0] := 2.584313;
   DATA[2440,1] := 867.1327;
   DATA[2440,2] := 2.0;
   DATA[2440,3] := 2.0;
   DATA[2440,4] := 262.3366;
   DATA[2440,5] := 8.395155;
   DATA[2440,6] := 329.7103;
   DATA[2440,7] := 2.453337;
   DATA[2440,8] := 2.0;
   DATA[2440,9] := 2.0;
   DATA[2440,10] := 2.0;
   DATA[2440,11] := 19.69396;
   DATA[2440,12] := 2.206322;
   DATA[2440,13] := 822.4254;
   DATA[2440,14] := 1.0;
   DATA[2440,15] := 2.0;
   DATA[2440,16] := 1.0;
   DATA[2440,17] := 1.0;
   DATA[2440,18] := 1.0;
   DATA[2440,19] := 2.0;
   DATA[2440,20] := 148.808;
   DATA[2440,21] := 155.3448;
   DATA[2440,22] := 1.712748;
   DATA[2440,23] := 862.202;
   DATA[2440,24] := 2.0;
   DATA[2440,25] := 2.0;
   DATA[2440,26] := 7.874135;
   DATA[2440,27] := 144.3732;
   DATA[2440,28] := 261.5996;
   DATA[2440,29] := 11.95847;
   DATA[2440,30] := 1.726609;
   DATA[2440,31] := 1.284873;
   DATA[2440,32] := 0.7353967;
   DATA[2440,33] := 0.309003;
   DATA[2440,34] := 2.0;
   DATA[2440,35] := 250.016;
   DATA[2440,36] := 1.585878;
   DATA[2440,37] := 188.8138;
   DATA[2440,38] := 0.000128152;
   DATA[2440,39] := 1.0;
   DATA[2440,40] := 1.0;
   DATA[2441,0] := 2.555488;
   DATA[2441,1] := 867.1719;
   DATA[2441,2] := 2.0;
   DATA[2441,3] := 2.0;
   DATA[2441,4] := 262.3366;
   DATA[2441,5] := 8.395155;
   DATA[2441,6] := 329.6334;
   DATA[2441,7] := 2.453337;
   DATA[2441,8] := 2.0;
   DATA[2441,9] := 2.0;
   DATA[2441,10] := 2.0;
   DATA[2441,11] := 19.69396;
   DATA[2441,12] := 2.206322;
   DATA[2441,13] := 822.1851;
   DATA[2441,14] := 1.0;
   DATA[2441,15] := 2.0;
   DATA[2441,16] := 1.0;
   DATA[2441,17] := 1.0;
   DATA[2441,18] := 1.0;
   DATA[2441,19] := 2.0;
   DATA[2441,20] := 148.808;
   DATA[2441,21] := 155.3448;
   DATA[2441,22] := 1.715952;
   DATA[2441,23] := 861.6252;
   DATA[2441,24] := 2.0;
   DATA[2441,25] := 2.0;
   DATA[2441,26] := 7.874135;
   DATA[2441,27] := 144.3732;
   DATA[2441,28] := 261.5996;
   DATA[2441,29] := 11.95847;
   DATA[2441,30] := 1.726609;
   DATA[2441,31] := 1.282183;
   DATA[2441,32] := 0.7353967;
   DATA[2441,33] := 0.309003;
   DATA[2441,34] := 2.0;
   DATA[2441,35] := 250.016;
   DATA[2441,36] := 1.585878;
   DATA[2441,37] := 188.8138;
   DATA[2441,38] := 0.000128152;
   DATA[2441,39] := 1.0;
   DATA[2441,40] := 1.0;
   DATA[2442,0] := 2.538513;
   DATA[2442,1] := 866.7794;
   DATA[2442,2] := 2.0;
   DATA[2442,3] := 2.0;
   DATA[2442,4] := 262.3366;
   DATA[2442,5] := 8.395155;
   DATA[2442,6] := 329.6334;
   DATA[2442,7] := 2.453337;
   DATA[2442,8] := 2.0;
   DATA[2442,9] := 2.0;
   DATA[2442,10] := 2.0;
   DATA[2442,11] := 19.69396;
   DATA[2442,12] := 2.206322;
   DATA[2442,13] := 822.2651;
   DATA[2442,14] := 1.0;
   DATA[2442,15] := 2.0;
   DATA[2442,16] := 1.0;
   DATA[2442,17] := 1.0;
   DATA[2442,18] := 1.0;
   DATA[2442,19] := 2.0;
   DATA[2442,20] := 148.808;
   DATA[2442,21] := 155.473;
   DATA[2442,22] := 1.716849;
   DATA[2442,23] := 861.7791;
   DATA[2442,24] := 2.0;
   DATA[2442,25] := 2.0;
   DATA[2442,26] := 7.874135;
   DATA[2442,27] := 144.3732;
   DATA[2442,28] := 261.5996;
   DATA[2442,29] := 11.95847;
   DATA[2442,30] := 1.726609;
   DATA[2442,31] := 1.290509;
   DATA[2442,32] := 0.7371892;
   DATA[2442,33] := 0.3084265;
   DATA[2442,34] := 2.0;
   DATA[2442,35] := 250.016;
   DATA[2442,36] := 1.585878;
   DATA[2442,37] := 188.8138;
   DATA[2442,38] := 0.000128152;
   DATA[2442,39] := 1.0;
   DATA[2442,40] := 1.0;
   DATA[2443,0] := 2.518656;
   DATA[2443,1] := 866.7794;
   DATA[2443,2] := 2.0;
   DATA[2443,3] := 2.0;
   DATA[2443,4] := 262.3045;
   DATA[2443,5] := 8.394514;
   DATA[2443,6] := 329.6334;
   DATA[2443,7] := 2.453337;
   DATA[2443,8] := 2.0;
   DATA[2443,9] := 2.0;
   DATA[2443,10] := 2.0;
   DATA[2443,11] := 19.72598;
   DATA[2443,12] := 2.206322;
   DATA[2443,13] := 822.3853;
   DATA[2443,14] := 1.0;
   DATA[2443,15] := 2.0;
   DATA[2443,16] := 1.0;
   DATA[2443,17] := 1.0;
   DATA[2443,18] := 1.0;
   DATA[2443,19] := 2.0;
   DATA[2443,20] := 148.808;
   DATA[2443,21] := 155.473;
   DATA[2443,22] := 1.718002;
   DATA[2443,23] := 861.7791;
   DATA[2443,24] := 2.0;
   DATA[2443,25] := 2.0;
   DATA[2443,26] := 7.874135;
   DATA[2443,27] := 144.3732;
   DATA[2443,28] := 261.5996;
   DATA[2443,29] := 11.95847;
   DATA[2443,30] := 1.728659;
   DATA[2443,31] := 1.295248;
   DATA[2443,32] := 0.7383414;
   DATA[2443,33] := 0.3084265;
   DATA[2443,34] := 2.0;
   DATA[2443,35] := 250.016;
   DATA[2443,36] := 1.746067;
   DATA[2443,37] := 188.8939;
   DATA[2443,38] := 0.000128152;
   DATA[2443,39] := 1.0;
   DATA[2443,40] := 1.0;
   DATA[2444,0] := 2.503603;
   DATA[2444,1] := 866.8579;
   DATA[2444,2] := 2.0;
   DATA[2444,3] := 2.0;
   DATA[2444,4] := 262.3045;
   DATA[2444,5] := 8.392271;
   DATA[2444,6] := 329.6334;
   DATA[2444,7] := 2.453337;
   DATA[2444,8] := 2.0;
   DATA[2444,9] := 2.0;
   DATA[2444,10] := 2.0;
   DATA[2444,11] := 19.74838;
   DATA[2444,12] := 2.207347;
   DATA[2444,13] := 822.3853;
   DATA[2444,14] := 1.0;
   DATA[2444,15] := 2.0;
   DATA[2444,16] := 1.0;
   DATA[2444,17] := 1.0;
   DATA[2444,18] := 1.0;
   DATA[2444,19] := 2.0;
   DATA[2444,20] := 148.808;
   DATA[2444,21] := 155.473;
   DATA[2444,22] := 1.718002;
   DATA[2444,23] := 861.5868;
   DATA[2444,24] := 2.0;
   DATA[2444,25] := 2.0;
   DATA[2444,26] := 7.874135;
   DATA[2444,27] := 144.3732;
   DATA[2444,28] := 261.5996;
   DATA[2444,29] := 11.95847;
   DATA[2444,30] := 1.728659;
   DATA[2444,31] := 1.302165;
   DATA[2444,32] := 0.7383414;
   DATA[2444,33] := 0.3084265;
   DATA[2444,34] := 2.0;
   DATA[2444,35] := 250.1442;
   DATA[2444,36] := 1.746067;
   DATA[2444,37] := 189.0381;
   DATA[2444,38] := 0.000128152;
   DATA[2444,39] := 1.0;
   DATA[2444,40] := 1.0;
   DATA[2445,0] := 2.483426;
   DATA[2445,1] := 867.0542;
   DATA[2445,2] := 2.0;
   DATA[2445,3] := 2.0;
   DATA[2445,4] := 262.3045;
   DATA[2445,5] := 8.392271;
   DATA[2445,6] := 329.6334;
   DATA[2445,7] := 2.453337;
   DATA[2445,8] := 2.0;
   DATA[2445,9] := 2.0;
   DATA[2445,10] := 2.0;
   DATA[2445,11] := 19.8028;
   DATA[2445,12] := 2.208244;
   DATA[2445,13] := 822.145;
   DATA[2445,14] := 1.0;
   DATA[2445,15] := 2.0;
   DATA[2445,16] := 1.0;
   DATA[2445,17] := 1.0;
   DATA[2445,18] := 1.0;
   DATA[2445,19] := 2.0;
   DATA[2445,20] := 148.808;
   DATA[2445,21] := 155.473;
   DATA[2445,22] := 1.718002;
   DATA[2445,23] := 862.0482;
   DATA[2445,24] := 2.0;
   DATA[2445,25] := 2.0;
   DATA[2445,26] := 7.874135;
   DATA[2445,27] := 144.3732;
   DATA[2445,28] := 261.5996;
   DATA[2445,29] := 11.95847;
   DATA[2445,30] := 1.728659;
   DATA[2445,31] := 1.299475;
   DATA[2445,32] := 0.7383414;
   DATA[2445,33] := 0.3084265;
   DATA[2445,34] := 2.0;
   DATA[2445,35] := 250.1442;
   DATA[2445,36] := 1.746067;
   DATA[2445,37] := 189.0381;
   DATA[2445,38] := 0.000128152;
   DATA[2445,39] := 1.0;
   DATA[2445,40] := 1.0;
   DATA[2446,0] := 2.472216;
   DATA[2446,1] := 867.2897;
   DATA[2446,2] := 2.0;
   DATA[2446,3] := 2.0;
   DATA[2446,4] := 262.3045;
   DATA[2446,5] := 8.392271;
   DATA[2446,6] := 329.6334;
   DATA[2446,7] := 2.453337;
   DATA[2446,8] := 2.0;
   DATA[2446,9] := 2.0;
   DATA[2446,10] := 2.0;
   DATA[2446,11] := 19.81881;
   DATA[2446,12] := 2.208244;
   DATA[2446,13] := 822.1851;
   DATA[2446,14] := 1.0;
   DATA[2446,15] := 2.0;
   DATA[2446,16] := 1.0;
   DATA[2446,17] := 1.0;
   DATA[2446,18] := 1.0;
   DATA[2446,19] := 2.0;
   DATA[2446,20] := 148.808;
   DATA[2446,21] := 155.473;
   DATA[2446,22] := 1.718515;
   DATA[2446,23] := 862.202;
   DATA[2446,24] := 2.0;
   DATA[2446,25] := 2.0;
   DATA[2446,26] := 7.874135;
   DATA[2446,27] := 144.5783;
   DATA[2446,28] := 261.5996;
   DATA[2446,29] := 11.95847;
   DATA[2446,30] := 1.728659;
   DATA[2446,31] := 1.291789;
   DATA[2446,32] := 0.7346286;
   DATA[2446,33] := 0.3084265;
   DATA[2446,34] := 2.0;
   DATA[2446,35] := 250.2724;
   DATA[2446,36] := 1.681991;
   DATA[2446,37] := 189.0861;
   DATA[2446,38] := 0.000128152;
   DATA[2446,39] := 1.0;
   DATA[2446,40] := 1.0;
   DATA[2447,0] := 2.45364;
   DATA[2447,1] := 867.1327;
   DATA[2447,2] := 2.0;
   DATA[2447,3] := 2.0;
   DATA[2447,4] := 262.3045;
   DATA[2447,5] := 8.392271;
   DATA[2447,6] := 329.6334;
   DATA[2447,7] := 2.453337;
   DATA[2447,8] := 2.0;
   DATA[2447,9] := 2.0;
   DATA[2447,10] := 2.0;
   DATA[2447,11] := 19.74198;
   DATA[2447,12] := 2.207347;
   DATA[2447,13] := 822.2651;
   DATA[2447,14] := 1.0;
   DATA[2447,15] := 2.0;
   DATA[2447,16] := 1.0;
   DATA[2447,17] := 1.0;
   DATA[2447,18] := 1.0;
   DATA[2447,19] := 2.0;
   DATA[2447,20] := 148.808;
   DATA[2447,21] := 155.473;
   DATA[2447,22] := 1.721078;
   DATA[2447,23] := 862.0482;
   DATA[2447,24] := 2.0;
   DATA[2447,25] := 2.0;
   DATA[2447,26] := 7.874135;
   DATA[2447,27] := 144.5783;
   DATA[2447,28] := 261.5996;
   DATA[2447,29] := 11.95847;
   DATA[2447,30] := 1.728659;
   DATA[2447,31] := 1.297041;
   DATA[2447,32] := 0.7346286;
   DATA[2447,33] := 0.3069532;
   DATA[2447,34] := 2.0;
   DATA[2447,35] := 250.2724;
   DATA[2447,36] := 1.665972;
   DATA[2447,37] := 189.1182;
   DATA[2447,38] := 0.000128152;
   DATA[2447,39] := 1.0;
   DATA[2447,40] := 1.0;
   DATA[2448,0] := 2.443071;
   DATA[2448,1] := 867.5252;
   DATA[2448,2] := 2.0;
   DATA[2448,3] := 2.0;
   DATA[2448,4] := 262.3045;
   DATA[2448,5] := 8.392271;
   DATA[2448,6] := 329.6334;
   DATA[2448,7] := 2.453337;
   DATA[2448,8] := 2.0;
   DATA[2448,9] := 2.0;
   DATA[2448,10] := 2.0;
   DATA[2448,11] := 19.68756;
   DATA[2448,12] := 2.206707;
   DATA[2448,13] := 822.0649;
   DATA[2448,14] := 1.0;
   DATA[2448,15] := 2.0;
   DATA[2448,16] := 1.0;
   DATA[2448,17] := 1.0;
   DATA[2448,18] := 1.0;
   DATA[2448,19] := 2.0;
   DATA[2448,20] := 148.808;
   DATA[2448,21] := 155.473;
   DATA[2448,22] := 1.721078;
   DATA[2448,23] := 862.2789;
   DATA[2448,24] := 2.0;
   DATA[2448,25] := 2.0;
   DATA[2448,26] := 7.874135;
   DATA[2448,27] := 144.5783;
   DATA[2448,28] := 261.5996;
   DATA[2448,29] := 11.95847;
   DATA[2448,30] := 1.728659;
   DATA[2448,31] := 1.295376;
   DATA[2448,32] := 0.7346286;
   DATA[2448,33] := 0.3069532;
   DATA[2448,34] := 2.0;
   DATA[2448,35] := 250.2724;
   DATA[2448,36] := 1.665972;
   DATA[2448,37] := 189.1182;
   DATA[2448,38] := 0.000128152;
   DATA[2448,39] := 1.0;
   DATA[2448,40] := 1.0;
   DATA[2449,0] := 2.427057;
   DATA[2449,1] := 867.5645;
   DATA[2449,2] := 2.0;
   DATA[2449,3] := 2.0;
   DATA[2449,4] := 262.3045;
   DATA[2449,5] := 8.392271;
   DATA[2449,6] := 329.6334;
   DATA[2449,7] := 2.453337;
   DATA[2449,8] := 2.0;
   DATA[2449,9] := 2.0;
   DATA[2449,10] := 2.0;
   DATA[2449,11] := 19.68756;
   DATA[2449,12] := 2.206707;
   DATA[2449,13] := 822.2651;
   DATA[2449,14] := 1.0;
   DATA[2449,15] := 2.0;
   DATA[2449,16] := 1.0;
   DATA[2449,17] := 1.0;
   DATA[2449,18] := 1.0;
   DATA[2449,19] := 2.0;
   DATA[2449,20] := 148.808;
   DATA[2449,21] := 155.473;
   DATA[2449,22] := 1.717874;
   DATA[2449,23] := 862.4327;
   DATA[2449,24] := 2.0;
   DATA[2449,25] := 2.0;
   DATA[2449,26] := 7.874135;
   DATA[2449,27] := 144.5783;
   DATA[2449,28] := 261.5996;
   DATA[2449,29] := 11.95847;
   DATA[2449,30] := 1.729172;
   DATA[2449,31] := 1.296529;
   DATA[2449,32] := 0.7346286;
   DATA[2449,33] := 0.3069532;
   DATA[2449,34] := 2.0;
   DATA[2449,35] := 250.2724;
   DATA[2449,36] := 1.665972;
   DATA[2449,37] := 189.1182;
   DATA[2449,38] := 0.000128152;
   DATA[2449,39] := 1.0;
   DATA[2449,40] := 1.0;
   DATA[2450,0] := 2.427057;
   DATA[2450,1] := 867.6429;
   DATA[2450,2] := 2.0;
   DATA[2450,3] := 2.0;
   DATA[2450,4] := 262.3045;
   DATA[2450,5] := 8.392271;
   DATA[2450,6] := 329.6334;
   DATA[2450,7] := 2.455003;
   DATA[2450,8] := 2.0;
   DATA[2450,9] := 2.0;
   DATA[2450,10] := 2.0;
   DATA[2450,11] := 19.68756;
   DATA[2450,12] := 2.206707;
   DATA[2450,13] := 821.9847;
   DATA[2450,14] := 1.0;
   DATA[2450,15] := 2.0;
   DATA[2450,16] := 1.0;
   DATA[2450,17] := 1.0;
   DATA[2450,18] := 1.0;
   DATA[2450,19] := 2.0;
   DATA[2450,20] := 148.808;
   DATA[2450,21] := 155.473;
   DATA[2450,22] := 1.717105;
   DATA[2450,23] := 862.5865;
   DATA[2450,24] := 2.0;
   DATA[2450,25] := 2.0;
   DATA[2450,26] := 7.874135;
   DATA[2450,27] := 144.5783;
   DATA[2450,28] := 261.5996;
   DATA[2450,29] := 11.95847;
   DATA[2450,30] := 1.729172;
   DATA[2450,31] := 1.290252;
   DATA[2450,32] := 0.7346286;
   DATA[2450,33] := 0.3069532;
   DATA[2450,34] := 2.0;
   DATA[2450,35] := 250.2724;
   DATA[2450,36] := 1.665972;
   DATA[2450,37] := 188.958;
   DATA[2450,38] := 0.000128152;
   DATA[2450,39] := 1.0;
   DATA[2450,40] := 1.0;
   DATA[2451,0] := 2.434744;
   DATA[2451,1] := 867.5252;
   DATA[2451,2] := 2.0;
   DATA[2451,3] := 2.0;
   DATA[2451,4] := 262.3045;
   DATA[2451,5] := 8.392271;
   DATA[2451,6] := 329.6334;
   DATA[2451,7] := 2.456412;
   DATA[2451,8] := 2.0;
   DATA[2451,9] := 2.0;
   DATA[2451,10] := 2.0;
   DATA[2451,11] := 19.68756;
   DATA[2451,12] := 2.206707;
   DATA[2451,13] := 822.4654;
   DATA[2451,14] := 1.0;
   DATA[2451,15] := 2.0;
   DATA[2451,16] := 1.0;
   DATA[2451,17] := 1.0;
   DATA[2451,18] := 1.0;
   DATA[2451,19] := 2.0;
   DATA[2451,20] := 148.808;
   DATA[2451,21] := 155.473;
   DATA[2451,22] := 1.717105;
   DATA[2451,23] := 862.7403;
   DATA[2451,24] := 2.0;
   DATA[2451,25] := 2.0;
   DATA[2451,26] := 7.874135;
   DATA[2451,27] := 144.5783;
   DATA[2451,28] := 261.5996;
   DATA[2451,29] := 11.95847;
   DATA[2451,30] := 1.729172;
   DATA[2451,31] := 1.273473;
   DATA[2451,32] := 0.7359089;
   DATA[2451,33] := 0.3069532;
   DATA[2451,34] := 2.0;
   DATA[2451,35] := 250.1602;
   DATA[2451,36] := 1.665972;
   DATA[2451,37] := 188.8618;
   DATA[2451,38] := 0.000128152;
   DATA[2451,39] := 1.0;
   DATA[2451,40] := 1.0;
   DATA[2452,0] := 2.468693;
   DATA[2452,1] := 867.6429;
   DATA[2452,2] := 2.0;
   DATA[2452,3] := 2.0;
   DATA[2452,4] := 262.3045;
   DATA[2452,5] := 8.393232;
   DATA[2452,6] := 329.6334;
   DATA[2452,7] := 2.456412;
   DATA[2452,8] := 2.0;
   DATA[2452,9] := 2.0;
   DATA[2452,10] := 2.0;
   DATA[2452,11] := 19.70997;
   DATA[2452,12] := 2.206707;
   DATA[2452,13] := 822.2651;
   DATA[2452,14] := 1.0;
   DATA[2452,15] := 2.0;
   DATA[2452,16] := 1.0;
   DATA[2452,17] := 1.0;
   DATA[2452,18] := 1.0;
   DATA[2452,19] := 2.0;
   DATA[2452,20] := 148.808;
   DATA[2452,21] := 155.473;
   DATA[2452,22] := 1.719027;
   DATA[2452,23] := 862.971;
   DATA[2452,24] := 2.0;
   DATA[2452,25] := 2.0;
   DATA[2452,26] := 7.874135;
   DATA[2452,27] := 144.5783;
   DATA[2452,28] := 261.5996;
   DATA[2452,29] := 11.95847;
   DATA[2452,30] := 1.725455;
   DATA[2452,31] := 1.265531;
   DATA[2452,32] := 0.7359089;
   DATA[2452,33] := 0.3084905;
   DATA[2452,34] := 2.0;
   DATA[2452,35] := 249.9039;
   DATA[2452,36] := 1.665972;
   DATA[2452,37] := 188.8618;
   DATA[2452,38] := 0.000128152;
   DATA[2452,39] := 1.0;
   DATA[2452,40] := 1.0;
   DATA[2453,0] := 2.519937;
   DATA[2453,1] := 867.8392;
   DATA[2453,2] := 2.0;
   DATA[2453,3] := 2.0;
   DATA[2453,4] := 262.3045;
   DATA[2453,5] := 8.396116;
   DATA[2453,6] := 329.6334;
   DATA[2453,7] := 2.456412;
   DATA[2453,8] := 2.0;
   DATA[2453,9] := 2.0;
   DATA[2453,10] := 2.0;
   DATA[2453,11] := 19.70997;
   DATA[2453,12] := 2.208244;
   DATA[2453,13] := 822.5455;
   DATA[2453,14] := 1.0;
   DATA[2453,15] := 2.0;
   DATA[2453,16] := 1.0;
   DATA[2453,17] := 1.0;
   DATA[2453,18] := 1.0;
   DATA[2453,19] := 2.0;
   DATA[2453,20] := 148.808;
   DATA[2453,21] := 155.473;
   DATA[2453,22] := 1.719027;
   DATA[2453,23] := 863.1248;
   DATA[2453,24] := 2.0;
   DATA[2453,25] := 2.0;
   DATA[2453,26] := 7.874135;
   DATA[2453,27] := 144.5783;
   DATA[2453,28] := 261.5996;
   DATA[2453,29] := 11.95847;
   DATA[2453,30] := 1.724942;
   DATA[2453,31] := 1.256052;
   DATA[2453,32] := 0.7359089;
   DATA[2453,33] := 0.3084905;
   DATA[2453,34] := 2.0;
   DATA[2453,35] := 249.9039;
   DATA[2453,36] := 1.69801;
   DATA[2453,37] := 188.8618;
   DATA[2453,38] := 0.000128152;
   DATA[2453,39] := 1.0;
   DATA[2453,40] := 1.0;
   DATA[2454,0] := 2.555168;
   DATA[2454,1] := 867.9177;
   DATA[2454,2] := 2.0;
   DATA[2454,3] := 2.0;
   DATA[2454,4] := 262.3045;
   DATA[2454,5] := 8.396116;
   DATA[2454,6] := 329.6334;
   DATA[2454,7] := 2.456412;
   DATA[2454,8] := 2.0;
   DATA[2454,9] := 2.0;
   DATA[2454,10] := 2.0;
   DATA[2454,11] := 19.65235;
   DATA[2454,12] := 2.208244;
   DATA[2454,13] := 822.2651;
   DATA[2454,14] := 1.0;
   DATA[2454,15] := 2.0;
   DATA[2454,16] := 1.0;
   DATA[2454,17] := 1.0;
   DATA[2454,18] := 1.0;
   DATA[2454,19] := 2.0;
   DATA[2454,20] := 148.808;
   DATA[2454,21] := 155.473;
   DATA[2454,22] := 1.717874;
   DATA[2454,23] := 863.5862;
   DATA[2454,24] := 2.0;
   DATA[2454,25] := 2.0;
   DATA[2454,26] := 7.874135;
   DATA[2454,27] := 144.5783;
   DATA[2454,28] := 261.5996;
   DATA[2454,29] := 11.95847;
   DATA[2454,30] := 1.724942;
   DATA[2454,31] := 1.264634;
   DATA[2454,32] := 0.7359089;
   DATA[2454,33] := 0.3084905;
   DATA[2454,34] := 2.0;
   DATA[2454,35] := 249.9039;
   DATA[2454,36] := 1.762086;
   DATA[2454,37] := 188.8618;
   DATA[2454,38] := 0.000128152;
   DATA[2454,39] := 1.0;
   DATA[2454,40] := 1.0;
   DATA[2455,0] := 2.595522;
   DATA[2455,1] := 868.114;
   DATA[2455,2] := 2.0;
   DATA[2455,3] := 2.0;
   DATA[2455,4] := 262.3045;
   DATA[2455,5] := 8.396116;
   DATA[2455,6] := 329.6334;
   DATA[2455,7] := 2.456412;
   DATA[2455,8] := 2.0;
   DATA[2455,9] := 2.0;
   DATA[2455,10] := 2.0;
   DATA[2455,11] := 19.65235;
   DATA[2455,12] := 2.208244;
   DATA[2455,13] := 822.5856;
   DATA[2455,14] := 1.0;
   DATA[2455,15] := 2.0;
   DATA[2455,16] := 1.0;
   DATA[2455,17] := 1.0;
   DATA[2455,18] := 1.0;
   DATA[2455,19] := 2.0;
   DATA[2455,20] := 148.808;
   DATA[2455,21] := 155.473;
   DATA[2455,22] := 1.715183;
   DATA[2455,23] := 863.3555;
   DATA[2455,24] := 2.0;
   DATA[2455,25] := 2.0;
   DATA[2455,26] := 7.874135;
   DATA[2455,27] := 144.5783;
   DATA[2455,28] := 261.5996;
   DATA[2455,29] := 11.95847;
   DATA[2455,30] := 1.724942;
   DATA[2455,31] := 1.277187;
   DATA[2455,32] := 0.7359089;
   DATA[2455,33] := 0.3084905;
   DATA[2455,34] := 2.0;
   DATA[2455,35] := 249.9039;
   DATA[2455,36] := 1.762086;
   DATA[2455,37] := 188.8618;
   DATA[2455,38] := 0.000128152;
   DATA[2455,39] := 1.0;
   DATA[2455,40] := 1.0;
   DATA[2456,0] := 2.624347;
   DATA[2456,1] := 868.3495;
   DATA[2456,2] := 2.0;
   DATA[2456,3] := 2.0;
   DATA[2456,4] := 262.3045;
   DATA[2456,5] := 8.396116;
   DATA[2456,6] := 329.6334;
   DATA[2456,7] := 2.456412;
   DATA[2456,8] := 2.0;
   DATA[2456,9] := 2.0;
   DATA[2456,10] := 2.0;
   DATA[2456,11] := 19.65235;
   DATA[2456,12] := 2.208884;
   DATA[2456,13] := 822.2251;
   DATA[2456,14] := 1.0;
   DATA[2456,15] := 2.0;
   DATA[2456,16] := 1.0;
   DATA[2456,17] := 1.0;
   DATA[2456,18] := 1.0;
   DATA[2456,19] := 2.0;
   DATA[2456,20] := 148.808;
   DATA[2456,21] := 155.4217;
   DATA[2456,22] := 1.714029;
   DATA[2456,23] := 863.6247;
   DATA[2456,24] := 2.0;
   DATA[2456,25] := 2.0;
   DATA[2456,26] := 7.874135;
   DATA[2456,27] := 144.5783;
   DATA[2456,28] := 261.5996;
   DATA[2456,29] := 11.95847;
   DATA[2456,30] := 1.724942;
   DATA[2456,31] := 1.288587;
   DATA[2456,32] := 0.7351407;
   DATA[2456,33] := 0.3084905;
   DATA[2456,34] := 2.0;
   DATA[2456,35] := 250.1442;
   DATA[2456,36] := 1.762086;
   DATA[2456,37] := 188.8618;
   DATA[2456,38] := 0.000128152;
   DATA[2456,39] := 1.0;
   DATA[2456,40] := 1.0;
   DATA[2457,0] := 2.647407;
   DATA[2457,1] := 867.957;
   DATA[2457,2] := 2.0;
   DATA[2457,3] := 2.0;
   DATA[2457,4] := 262.3045;
   DATA[2457,5] := 8.396116;
   DATA[2457,6] := 329.6334;
   DATA[2457,7] := 2.455131;
   DATA[2457,8] := 2.0;
   DATA[2457,9] := 2.0;
   DATA[2457,10] := 2.0;
   DATA[2457,11] := 19.67796;
   DATA[2457,12] := 2.209269;
   DATA[2457,13] := 822.5455;
   DATA[2457,14] := 1.0;
   DATA[2457,15] := 2.0;
   DATA[2457,16] := 1.0;
   DATA[2457,17] := 1.0;
   DATA[2457,18] := 1.0;
   DATA[2457,19] := 2.0;
   DATA[2457,20] := 148.808;
   DATA[2457,21] := 155.4217;
   DATA[2457,22] := 1.713901;
   DATA[2457,23] := 864.163;
   DATA[2457,24] := 2.0;
   DATA[2457,25] := 2.0;
   DATA[2457,26] := 7.874135;
   DATA[2457,27] := 144.5783;
   DATA[2457,28] := 261.5996;
   DATA[2457,29] := 11.95847;
   DATA[2457,30] := 1.724942;
   DATA[2457,31] := 1.301396;
   DATA[2457,32] := 0.7351407;
   DATA[2457,33] := 0.3084905;
   DATA[2457,34] := 2.0;
   DATA[2457,35] := 250.1442;
   DATA[2457,36] := 1.826162;
   DATA[2457,37] := 188.8618;
   DATA[2457,38] := 0.000128152;
   DATA[2457,39] := 1.0;
   DATA[2457,40] := 1.0;
   DATA[2458,0] := 2.658937;
   DATA[2458,1] := 868.3495;
   DATA[2458,2] := 2.0;
   DATA[2458,3] := 2.0;
   DATA[2458,4] := 262.3045;
   DATA[2458,5] := 8.396116;
   DATA[2458,6] := 329.6334;
   DATA[2458,7] := 2.455131;
   DATA[2458,8] := 2.0;
   DATA[2458,9] := 2.0;
   DATA[2458,10] := 2.0;
   DATA[2458,11] := 19.70037;
   DATA[2458,12] := 2.209653;
   DATA[2458,13] := 822.5455;
   DATA[2458,14] := 1.0;
   DATA[2458,15] := 2.0;
   DATA[2458,16] := 1.0;
   DATA[2458,17] := 1.0;
   DATA[2458,18] := 1.0;
   DATA[2458,19] := 2.0;
   DATA[2458,20] := 148.808;
   DATA[2458,21] := 155.2166;
   DATA[2458,22] := 1.713901;
   DATA[2458,23] := 864.3168;
   DATA[2458,24] := 2.0;
   DATA[2458,25] := 2.0;
   DATA[2458,26] := 7.874135;
   DATA[2458,27] := 144.5783;
   DATA[2458,28] := 261.5996;
   DATA[2458,29] := 11.95847;
   DATA[2458,30] := 1.724942;
   DATA[2458,31] := 1.302037;
   DATA[2458,32] := 0.7351407;
   DATA[2458,33] := 0.3084905;
   DATA[2458,34] := 2.0;
   DATA[2458,35] := 250.1442;
   DATA[2458,36] := 1.826162;
   DATA[2458,37] := 188.8618;
   DATA[2458,38] := 0.000128152;
   DATA[2458,39] := 1.0;
   DATA[2458,40] := 1.0;
   DATA[2459,0] := 2.659578;
   DATA[2459,1] := 868.428;
   DATA[2459,2] := 2.0;
   DATA[2459,3] := 2.0;
   DATA[2459,4] := 262.3045;
   DATA[2459,5] := 8.396116;
   DATA[2459,6] := 329.6334;
   DATA[2459,7] := 2.452696;
   DATA[2459,8] := 2.0;
   DATA[2459,9] := 2.0;
   DATA[2459,10] := 2.0;
   DATA[2459,11] := 19.70037;
   DATA[2459,12] := 2.21055;
   DATA[2459,13] := 822.8259;
   DATA[2459,14] := 1.0;
   DATA[2459,15] := 2.0;
   DATA[2459,16] := 1.0;
   DATA[2459,17] := 1.0;
   DATA[2459,18] := 1.0;
   DATA[2459,19] := 2.0;
   DATA[2459,20] := 148.808;
   DATA[2459,21] := 155.2166;
   DATA[2459,22] := 1.71467;
   DATA[2459,23] := 864.5091;
   DATA[2459,24] := 2.0;
   DATA[2459,25] := 2.0;
   DATA[2459,26] := 7.874135;
   DATA[2459,27] := 144.5783;
   DATA[2459,28] := 261.5996;
   DATA[2459,29] := 11.95847;
   DATA[2459,30] := 1.726352;
   DATA[2459,31] := 1.302037;
   DATA[2459,32] := 0.7351407;
   DATA[2459,33] := 0.3084905;
   DATA[2459,34] := 2.0;
   DATA[2459,35] := 250.1442;
   DATA[2459,36] := 1.826162;
   DATA[2459,37] := 188.8618;
   DATA[2459,38] := 0.000128152;
   DATA[2459,39] := 1.0;
   DATA[2459,40] := 1.0;
   DATA[2460,0] := 2.640361;
   DATA[2460,1] := 868.6243;
   DATA[2460,2] := 2.0;
   DATA[2460,3] := 2.0;
   DATA[2460,4] := 262.3045;
   DATA[2460,5] := 8.396116;
   DATA[2460,6] := 329.6334;
   DATA[2460,7] := 2.452696;
   DATA[2460,8] := 2.0;
   DATA[2460,9] := 2.0;
   DATA[2460,10] := 2.0;
   DATA[2460,11] := 19.70037;
   DATA[2460,12] := 2.21055;
   DATA[2460,13] := 822.7858;
   DATA[2460,14] := 1.0;
   DATA[2460,15] := 2.0;
   DATA[2460,16] := 1.0;
   DATA[2460,17] := 1.0;
   DATA[2460,18] := 1.0;
   DATA[2460,19] := 2.0;
   DATA[2460,20] := 148.808;
   DATA[2460,21] := 155.2166;
   DATA[2460,22] := 1.71467;
   DATA[2460,23] := 864.5475;
   DATA[2460,24] := 2.0;
   DATA[2460,25] := 2.0;
   DATA[2460,26] := 7.874135;
   DATA[2460,27] := 144.5783;
   DATA[2460,28] := 261.5996;
   DATA[2460,29] := 11.95847;
   DATA[2460,30] := 1.726737;
   DATA[2460,31] := 1.295632;
   DATA[2460,32] := 0.7351407;
   DATA[2460,33] := 0.3084905;
   DATA[2460,34] := 2.0;
   DATA[2460,35] := 250.1442;
   DATA[2460,36] := 1.826162;
   DATA[2460,37] := 188.974;
   DATA[2460,38] := 0.000128152;
   DATA[2460,39] := 1.0;
   DATA[2460,40] := 1.0;
   DATA[2461,0] := 2.624027;
   DATA[2461,1] := 868.7421;
   DATA[2461,2] := 2.0;
   DATA[2461,3] := 2.0;
   DATA[2461,4] := 262.3045;
   DATA[2461,5] := 8.396116;
   DATA[2461,6] := 329.6334;
   DATA[2461,7] := 2.452696;
   DATA[2461,8] := 2.0;
   DATA[2461,9] := 2.0;
   DATA[2461,10] := 2.0;
   DATA[2461,11] := 19.70037;
   DATA[2461,12] := 2.21055;
   DATA[2461,13] := 822.866;
   DATA[2461,14] := 1.0;
   DATA[2461,15] := 2.0;
   DATA[2461,16] := 1.0;
   DATA[2461,17] := 1.0;
   DATA[2461,18] := 1.0;
   DATA[2461,19] := 2.0;
   DATA[2461,20] := 148.808;
   DATA[2461,21] := 155.2166;
   DATA[2461,22] := 1.71467;
   DATA[2461,23] := 864.8552;
   DATA[2461,24] := 2.0;
   DATA[2461,25] := 2.0;
   DATA[2461,26] := 7.874135;
   DATA[2461,27] := 144.5783;
   DATA[2461,28] := 261.5996;
   DATA[2461,29] := 11.95847;
   DATA[2461,30] := 1.726737;
   DATA[2461,31] := 1.30114;
   DATA[2461,32] := 0.7351407;
   DATA[2461,33] := 0.3084905;
   DATA[2461,34] := 2.0;
   DATA[2461,35] := 250.1442;
   DATA[2461,36] := 1.69801;
   DATA[2461,37] := 188.974;
   DATA[2461,38] := 0.000128152;
   DATA[2461,39] := 1.0;
   DATA[2461,40] := 1.0;
   DATA[2462,0] := 2.618903;
   DATA[2462,1] := 868.271;
   DATA[2462,2] := 2.0;
   DATA[2462,3] := 2.0;
   DATA[2462,4] := 262.3045;
   DATA[2462,5] := 8.396116;
   DATA[2462,6] := 329.6334;
   DATA[2462,7] := 2.452696;
   DATA[2462,8] := 2.0;
   DATA[2462,9] := 2.0;
   DATA[2462,10] := 2.0;
   DATA[2462,11] := 19.70037;
   DATA[2462,12] := 2.209653;
   DATA[2462,13] := 823.3867;
   DATA[2462,14] := 1.0;
   DATA[2462,15] := 2.0;
   DATA[2462,16] := 1.0;
   DATA[2462,17] := 1.0;
   DATA[2462,18] := 1.0;
   DATA[2462,19] := 2.0;
   DATA[2462,20] := 148.808;
   DATA[2462,21] := 155.2166;
   DATA[2462,22] := 1.71467;
   DATA[2462,23] := 865.0474;
   DATA[2462,24] := 2.0;
   DATA[2462,25] := 2.0;
   DATA[2462,26] := 7.874135;
   DATA[2462,27] := 144.5783;
   DATA[2462,28] := 261.5996;
   DATA[2462,29] := 11.95847;
   DATA[2462,30] := 1.726737;
   DATA[2462,31] := 1.302293;
   DATA[2462,32] := 0.7351407;
   DATA[2462,33] := 0.3084905;
   DATA[2462,34] := 2.0;
   DATA[2462,35] := 250.1442;
   DATA[2462,36] := 1.69801;
   DATA[2462,37] := 189.0541;
   DATA[2462,38] := 0.000128152;
   DATA[2462,39] := 1.0;
   DATA[2462,40] := 1.0;
   DATA[2463,0] := 2.612818;
   DATA[2463,1] := 868.2318;
   DATA[2463,2] := 2.0;
   DATA[2463,3] := 2.0;
   DATA[2463,4] := 262.3045;
   DATA[2463,5] := 8.396116;
   DATA[2463,6] := 329.6334;
   DATA[2463,7] := 2.452696;
   DATA[2463,8] := 2.0;
   DATA[2463,9] := 2.0;
   DATA[2463,10] := 2.0;
   DATA[2463,11] := 19.70037;
   DATA[2463,12] := 2.209653;
   DATA[2463,13] := 823.3466;
   DATA[2463,14] := 1.0;
   DATA[2463,15] := 2.0;
   DATA[2463,16] := 1.0;
   DATA[2463,17] := 1.0;
   DATA[2463,18] := 1.0;
   DATA[2463,19] := 2.0;
   DATA[2463,20] := 148.808;
   DATA[2463,21] := 155.2166;
   DATA[2463,22] := 1.71467;
   DATA[2463,23] := 865.8549;
   DATA[2463,24] := 2.0;
   DATA[2463,25] := 2.0;
   DATA[2463,26] := 7.874135;
   DATA[2463,27] := 144.5783;
   DATA[2463,28] := 261.5996;
   DATA[2463,29] := 11.95847;
   DATA[2463,30] := 1.726865;
   DATA[2463,31] := 1.306264;
   DATA[2463,32] := 0.7351407;
   DATA[2463,33] := 0.3084905;
   DATA[2463,34] := 2.0;
   DATA[2463,35] := 250.1442;
   DATA[2463,36] := 1.69801;
   DATA[2463,37] := 189.0541;
   DATA[2463,38] := 0.000128152;
   DATA[2463,39] := 1.0;
   DATA[2463,40] := 1.0;
   DATA[2464,0] := 2.589757;
   DATA[2464,1] := 868.3102;
   DATA[2464,2] := 2.0;
   DATA[2464,3] := 2.0;
   DATA[2464,4] := 262.3045;
   DATA[2464,5] := 8.396116;
   DATA[2464,6] := 329.6334;
   DATA[2464,7] := 2.452696;
   DATA[2464,8] := 2.0;
   DATA[2464,9] := 2.0;
   DATA[2464,10] := 2.0;
   DATA[2464,11] := 19.70357;
   DATA[2464,12] := 2.209653;
   DATA[2464,13] := 823.7471;
   DATA[2464,14] := 1.0;
   DATA[2464,15] := 2.0;
   DATA[2464,16] := 1.0;
   DATA[2464,17] := 1.0;
   DATA[2464,18] := 1.0;
   DATA[2464,19] := 2.0;
   DATA[2464,20] := 148.808;
   DATA[2464,21] := 155.2166;
   DATA[2464,22] := 1.71467;
   DATA[2464,23] := 865.9318;
   DATA[2464,24] := 2.0;
   DATA[2464,25] := 2.0;
   DATA[2464,26] := 7.874135;
   DATA[2464,27] := 144.5783;
   DATA[2464,28] := 261.5996;
   DATA[2464,29] := 11.95847;
   DATA[2464,30] := 1.726865;
   DATA[2464,31] := 1.310747;
   DATA[2464,32] := 0.7351407;
   DATA[2464,33] := 0.3084905;
   DATA[2464,34] := 2.0;
   DATA[2464,35] := 250.1442;
   DATA[2464,36] := 1.69801;
   DATA[2464,37] := 189.0541;
   DATA[2464,38] := 0.000128152;
   DATA[2464,39] := 1.0;
   DATA[2464,40] := 1.0;
   DATA[2465,0] := 2.570541;
   DATA[2465,1] := 868.271;
   DATA[2465,2] := 2.0;
   DATA[2465,3] := 2.0;
   DATA[2465,4] := 262.3045;
   DATA[2465,5] := 8.393873;
   DATA[2465,6] := 329.6334;
   DATA[2465,7] := 2.452312;
   DATA[2465,8] := 2.0;
   DATA[2465,9] := 2.0;
   DATA[2465,10] := 2.0;
   DATA[2465,11] := 19.72598;
   DATA[2465,12] := 2.209653;
   DATA[2465,13] := 824.0676;
   DATA[2465,14] := 1.0;
   DATA[2465,15] := 2.0;
   DATA[2465,16] := 1.0;
   DATA[2465,17] := 1.0;
   DATA[2465,18] := 1.0;
   DATA[2465,19] := 2.0;
   DATA[2465,20] := 148.808;
   DATA[2465,21] := 155.2166;
   DATA[2465,22] := 1.716592;
   DATA[2465,23] := 866.0472;
   DATA[2465,24] := 2.0;
   DATA[2465,25] := 2.0;
   DATA[2465,26] := 7.874135;
   DATA[2465,27] := 144.5783;
   DATA[2465,28] := 261.5996;
   DATA[2465,29] := 11.95847;
   DATA[2465,30] := 1.726865;
   DATA[2465,31] := 1.296529;
   DATA[2465,32] := 0.7351407;
   DATA[2465,33] := 0.3084905;
   DATA[2465,34] := 2.0;
   DATA[2465,35] := 250.1442;
   DATA[2465,36] := 1.69801;
   DATA[2465,37] := 189.0541;
   DATA[2465,38] := 0.000128152;
   DATA[2465,39] := 1.0;
   DATA[2465,40] := 1.0;
   DATA[2466,0] := 2.550684;
   DATA[2466,1] := 868.2318;
   DATA[2466,2] := 2.0;
   DATA[2466,3] := 2.0;
   DATA[2466,4] := 262.3045;
   DATA[2466,5] := 8.393873;
   DATA[2466,6] := 329.6334;
   DATA[2466,7] := 2.451927;
   DATA[2466,8] := 2.0;
   DATA[2466,9] := 2.0;
   DATA[2466,10] := 2.0;
   DATA[2466,11] := 19.74198;
   DATA[2466,12] := 2.208244;
   DATA[2466,13] := 824.2278;
   DATA[2466,14] := 1.0;
   DATA[2466,15] := 2.0;
   DATA[2466,16] := 1.0;
   DATA[2466,17] := 1.0;
   DATA[2466,18] := 1.0;
   DATA[2466,19] := 2.0;
   DATA[2466,20] := 148.808;
   DATA[2466,21] := 155.2166;
   DATA[2466,22] := 1.716592;
   DATA[2466,23] := 865.8165;
   DATA[2466,24] := 2.0;
   DATA[2466,25] := 2.0;
   DATA[2466,26] := 7.874135;
   DATA[2466,27] := 144.5783;
   DATA[2466,28] := 261.5996;
   DATA[2466,29] := 11.95847;
   DATA[2466,30] := 1.726609;
   DATA[2466,31] := 1.284488;
   DATA[2466,32] := 0.7352687;
   DATA[2466,33] := 0.3084905;
   DATA[2466,34] := 2.0;
   DATA[2466,35] := 250.1442;
   DATA[2466,36] := 1.69801;
   DATA[2466,37] := 188.8779;
   DATA[2466,38] := 0.000128152;
   DATA[2466,39] := 1.0;
   DATA[2466,40] := 1.0;
   DATA[2467,0] := 2.537232;
   DATA[2467,1] := 868.271;
   DATA[2467,2] := 2.0;
   DATA[2467,3] := 2.0;
   DATA[2467,4] := 262.3045;
   DATA[2467,5] := 8.393873;
   DATA[2467,6] := 329.6334;
   DATA[2467,7] := 2.451927;
   DATA[2467,8] := 2.0;
   DATA[2467,9] := 2.0;
   DATA[2467,10] := 2.0;
   DATA[2467,11] := 19.74198;
   DATA[2467,12] := 2.206963;
   DATA[2467,13] := 824.5482;
   DATA[2467,14] := 1.0;
   DATA[2467,15] := 2.0;
   DATA[2467,16] := 1.0;
   DATA[2467,17] := 1.0;
   DATA[2467,18] := 1.0;
   DATA[2467,19] := 2.0;
   DATA[2467,20] := 148.808;
   DATA[2467,21] := 155.2166;
   DATA[2467,22] := 1.716592;
   DATA[2467,23] := 866.5855;
   DATA[2467,24] := 2.0;
   DATA[2467,25] := 2.0;
   DATA[2467,26] := 7.874135;
   DATA[2467,27] := 144.5783;
   DATA[2467,28] := 261.5996;
   DATA[2467,29] := 11.95847;
   DATA[2467,30] := 1.725711;
   DATA[2467,31] := 1.281798;
   DATA[2467,32] := 0.7353967;
   DATA[2467,33] := 0.3084905;
   DATA[2467,34] := 2.0;
   DATA[2467,35] := 250.1442;
   DATA[2467,36] := 1.69801;
   DATA[2467,37] := 188.8458;
   DATA[2467,38] := 0.000128152;
   DATA[2467,39] := 1.0;
   DATA[2467,40] := 1.0;
   DATA[2468,0] := 2.520257;
   DATA[2468,1] := 867.9177;
   DATA[2468,2] := 2.0;
   DATA[2468,3] := 2.0;
   DATA[2468,4] := 262.3045;
   DATA[2468,5] := 8.393873;
   DATA[2468,6] := 329.6334;
   DATA[2468,7] := 2.451927;
   DATA[2468,8] := 2.0;
   DATA[2468,9] := 2.0;
   DATA[2468,10] := 2.0;
   DATA[2468,11] := 19.74198;
   DATA[2468,12] := 2.206963;
   DATA[2468,13] := 824.5883;
   DATA[2468,14] := 1.0;
   DATA[2468,15] := 2.0;
   DATA[2468,16] := 1.0;
   DATA[2468,17] := 1.0;
   DATA[2468,18] := 1.0;
   DATA[2468,19] := 2.0;
   DATA[2468,20] := 148.808;
   DATA[2468,21] := 155.2166;
   DATA[2468,22] := 1.716592;
   DATA[2468,23] := 866.3163;
   DATA[2468,24] := 2.0;
   DATA[2468,25] := 2.0;
   DATA[2468,26] := 7.874135;
   DATA[2468,27] := 144.5783;
   DATA[2468,28] := 261.5675;
   DATA[2468,29] := 11.95847;
   DATA[2468,30] := 1.725711;
   DATA[2468,31] := 1.274753;
   DATA[2468,32] := 0.7353967;
   DATA[2468,33] := 0.3084905;
   DATA[2468,34] := 2.0;
   DATA[2468,35] := 250.1442;
   DATA[2468,36] := 1.69801;
   DATA[2468,37] := 188.8458;
   DATA[2468,38] := 0.000128152;
   DATA[2468,39] := 1.0;
   DATA[2468,40] := 1.0;
   DATA[2469,0] := 2.502642;
   DATA[2469,1] := 867.5645;
   DATA[2469,2] := 2.0;
   DATA[2469,3] := 2.0;
   DATA[2469,4] := 262.3045;
   DATA[2469,5] := 8.393873;
   DATA[2469,6] := 329.8385;
   DATA[2469,7] := 2.451927;
   DATA[2469,8] := 2.0;
   DATA[2469,9] := 2.0;
   DATA[2469,10] := 2.0;
   DATA[2469,11] := 19.74198;
   DATA[2469,12] := 2.208756;
   DATA[2469,13] := 824.9888;
   DATA[2469,14] := 1.0;
   DATA[2469,15] := 2.0;
   DATA[2469,16] := 1.0;
   DATA[2469,17] := 1.0;
   DATA[2469,18] := 1.0;
   DATA[2469,19] := 2.0;
   DATA[2469,20] := 148.808;
   DATA[2469,21] := 155.2166;
   DATA[2469,22] := 1.716592;
   DATA[2469,23] := 866.6624;
   DATA[2469,24] := 2.0;
   DATA[2469,25] := 2.0;
   DATA[2469,26] := 7.874135;
   DATA[2469,27] := 144.5783;
   DATA[2469,28] := 261.5034;
   DATA[2469,29] := 11.95847;
   DATA[2469,30] := 1.725711;
   DATA[2469,31] := 1.271295;
   DATA[2469,32] := 0.7353967;
   DATA[2469,33] := 0.3084905;
   DATA[2469,34] := 2.0;
   DATA[2469,35] := 250.1442;
   DATA[2469,36] := 1.69801;
   DATA[2469,37] := 188.8458;
   DATA[2469,38] := 0.000128152;
   DATA[2469,39] := 1.0;
   DATA[2469,40] := 1.0;
   DATA[2470,0] := 2.482465;
   DATA[2470,1] := 866.8579;
   DATA[2470,2] := 2.0;
   DATA[2470,3] := 2.0;
   DATA[2470,4] := 262.3045;
   DATA[2470,5] := 8.393873;
   DATA[2470,6] := 329.8385;
   DATA[2470,7] := 2.451927;
   DATA[2470,8] := 2.0;
   DATA[2470,9] := 2.0;
   DATA[2470,10] := 2.0;
   DATA[2470,11] := 19.76759;
   DATA[2470,12] := 2.208756;
   DATA[2470,13] := 825.1891;
   DATA[2470,14] := 1.0;
   DATA[2470,15] := 2.0;
   DATA[2470,16] := 1.0;
   DATA[2470,17] := 1.0;
   DATA[2470,18] := 1.0;
   DATA[2470,19] := 2.0;
   DATA[2470,20] := 148.808;
   DATA[2470,21] := 155.2166;
   DATA[2470,22] := 1.716592;
   DATA[2470,23] := 866.97;
   DATA[2470,24] := 2.0;
   DATA[2470,25] := 2.0;
   DATA[2470,26] := 7.874135;
   DATA[2470,27] := 144.5783;
   DATA[2470,28] := 261.5034;
   DATA[2470,29] := 11.95847;
   DATA[2470,30] := 1.725711;
   DATA[2470,31] := 1.271423;
   DATA[2470,32] := 0.7353967;
   DATA[2470,33] := 0.3084905;
   DATA[2470,34] := 2.0;
   DATA[2470,35] := 250.1442;
